LIN {X 0.032,Y -167.550,Z 313.355,A 0.000,B 0.000,C 90.000,E1 243.896} C_DIS
LIN {X 0.046,Y -166.172,Z 313.345,A 0.000,B 0.000,C 90.000,E1 242.153} C_DIS
LIN {X 0.036,Y -162.944,Z 313.326,A 0.000,B 0.000,C 90.000,E1 238.663} C_DIS
LIN {X 0.014,Y -161.614,Z 313.316,A 0.000,B 0.000,C 90.000,E1 236.914} C_DIS
LIN {X -0.011,Y -159.142,Z 313.302,A 0.000,B 0.000,C 90.000,E1 234.276} C_DIS
LIN {X -0.001,Y -155.664,Z 313.277,A 0.000,B 0.000,C 90.000,E1 229.828} C_DIS
LIN {X 0.052,Y -151.932,Z 313.252,A 0.000,B 0.000,C 90.000,E1 225.324} C_DIS
LIN {X 0.066,Y -150.169,Z 313.237,A 0.000,B 0.000,C 90.000,E1 222.609} C_DIS
LIN {X -0.014,Y -146.946,Z 313.212,A 0.000,B 0.000,C 90.000,E1 218.096} C_DIS
LIN {X -0.026,Y -145.534,Z 313.196,A 0.000,B 0.000,C 90.000,E1 215.358} C_DIS
LIN {X 0.014,Y -142.931,Z 313.171,A 0.000,B 0.000,C 90.000,E1 210.747} C_DIS
LIN {X 0.013,Y -141.555,Z 313.150,A 0.000,B 0.000,C 90.000,E1 207.052} C_DIS
LIN {X 0.001,Y -139.407,Z 313.114,A 0.000,B 0.000,C 90.000,E1 200.556} C_DIS
LIN {X -0.077,Y -139.126,Z 313.104,A 0.000,B 0.000,C 90.000,E1 198.725} C_DIS
LIN {X -0.050,Y -138.351,Z 313.057,A 0.000,B 0.000,C 90.000,E1 190.310} C_DIS
LIN {X -0.062,Y -139.500,Z 313.005,A 0.000,B 0.000,C 90.000,E1 180.974} C_DIS
LIN {X 0.018,Y -141.125,Z 312.974,A 0.000,B 0.000,C 90.000,E1 175.355} C_DIS
LIN {X -0.029,Y -142.505,Z 312.959,A 0.000,B 0.000,C 90.000,E1 172.591} C_DIS
LIN {X 0.059,Y -144.762,Z 312.933,A 0.000,B 0.000,C 90.000,E1 167.937} C_DIS
LIN {X 0.008,Y -147.373,Z 312.913,A 0.000,B 0.000,C 90.000,E1 164.283} C_DIS
LIN {X 0.071,Y -150.702,Z 312.887,A 0.000,B 0.000,C 90.000,E1 159.699} C_DIS
LIN {X 0.013,Y -154.182,Z 312.867,A 0.000,B 0.000,C 90.000,E1 156.102} C_DIS
LIN {X -0.058,Y -157.618,Z 312.847,A 0.000,B 0.000,C 90.000,E1 152.538} C_DIS
LIN {X 0.030,Y -161.873,Z 312.828,A 0.000,B 0.000,C 90.000,E1 148.948} C_DIS
LIN {X 0.003,Y -166.064,Z 312.808,A 0.000,B 0.000,C 90.000,E1 145.435} C_DIS
LIN {X 0.004,Y -171.069,Z 312.789,A 0.000,B 0.000,C 90.000,E1 141.949} C_DIS
LIN {X 0.060,Y -175.942,Z 312.769,A 0.000,B 0.000,C 90.000,E1 138.485} C_DIS
LIN {X -0.080,Y -180.183,Z 312.755,A 0.000,B 0.000,C 90.000,E1 135.972} C_DIS
LIN {X -0.112,Y -185.599,Z 312.737,A 0.000,B 0.000,C 90.000,E1 132.609} C_DIS
LIN {X -0.062,Y -190.191,Z 312.723,A 0.000,B 0.000,C 90.000,E1 130.092} C_DIS
LIN {X -0.018,Y -197.520,Z 312.700,A 0.000,B 0.000,C 90.000,E1 125.964} C_DIS
LIN {X -0.040,Y -201.256,Z 312.689,A 0.000,B 0.000,C 90.000,E1 124.072} C_DIS
LIN {X 0.037,Y -201.982,Z 312.687,A 0.000,B 0.000,C 90.000,E1 123.627} C_DIS
LIN {X 0.021,Y -303.002,Z 312.687,A 0.000,B 0.000,C 90.000,E1 123.627} C_DIS
LIN {X 0.128,Y -307.334,Z 312.686,A 0.000,B 0.000,C 90.000,E1 123.499} C_DIS
LIN {X 0.193,Y -310.491,Z 312.685,A 0.000,B 0.000,C 90.000,E1 123.293} C_DIS
LIN {X -0.027,Y -314.159,Z 312.683,A 0.000,B 0.000,C 90.000,E1 122.959} C_DIS
LIN {X -0.196,Y -317.653,Z 312.680,A 0.000,B 0.000,C 90.000,E1 122.418} C_DIS
LIN {X -0.068,Y -320.195,Z 312.676,A 0.000,B 0.000,C 90.000,E1 121.750} C_DIS
LIN {X 0.051,Y -331.214,Z 312.660,A 0.000,B 0.000,C 90.000,E1 118.871} C_DIS
LIN {X -0.163,Y -343.646,Z 312.645,A 0.000,B 0.000,C 90.000,E1 116.104} C_DIS
LIN {X -0.044,Y -355.971,Z 312.631,A 0.000,B 0.000,C 90.000,E1 113.643} C_DIS
LIN {X 0.113,Y -369.589,Z 312.618,A 0.000,B 0.000,C 90.000,E1 111.227} C_DIS
LIN {X 0.003,Y -384.601,Z 312.605,A 0.000,B 0.000,C 90.000,E1 108.906} C_DIS
LIN {X 0.015,Y -401.116,Z 312.592,A 0.000,B 0.000,C 90.000,E1 106.622} C_DIS
LIN {X -0.074,Y -419.259,Z 312.580,A 0.000,B 0.000,C 90.000,E1 104.411} C_DIS
LIN {X 0.118,Y -438.973,Z 312.568,A 0.000,B 0.000,C 90.000,E1 102.243} C_DIS
LIN {X -0.205,Y -459.388,Z 312.557,A 0.000,B 0.000,C 90.000,E1 100.310} C_DIS
LIN {X -0.132,Y -482.952,Z 312.546,A 0.000,B 0.000,C 90.000,E1 98.276} C_DIS
LIN {X -0.206,Y -496.291,Z 312.540,A 0.000,B 0.000,C 90.000,E1 97.239} C_DIS
LIN {X 0.248,Y -500.118,Z 312.538,A 0.000,B 0.000,C 90.000,E1 96.777} C_DIS
LIN {X 0.104,Y -501.638,Z 312.536,A 0.000,B 0.000,C 90.000,E1 96.549} C_DIS
LIN {X 0.015,Y -502.770,Z 312.535,A 0.000,B 0.000,C 90.000,E1 96.315} C_DIS
LIN {X -0.190,Y -504.107,Z 312.532,A 0.000,B 0.000,C 90.000,E1 95.853} C_DIS
LIN {X 0.111,Y -504.399,Z 312.530,A 0.000,B 0.000,C 90.000,E1 95.334} C_DIS
LIN {X -0.127,Y -503.685,Z 312.527,A 0.000,B 0.000,C 90.000,E1 94.878} C_DIS
LIN {X 0.184,Y -501.840,Z 312.524,A 0.000,B 0.000,C 90.000,E1 94.359} C_DIS
LIN {X 0.067,Y -500.376,Z 312.523,A 0.000,B 0.000,C 90.000,E1 94.131} C_DIS
LIN {X 0.233,Y -494.896,Z 312.519,A 0.000,B 0.000,C 90.000,E1 93.383} C_DIS
LIN {X 0.203,Y -486.911,Z 312.514,A 0.000,B 0.000,C 90.000,E1 92.407} C_DIS
LIN {X -0.144,Y -470.368,Z 312.502,A 0.000,B 0.000,C 90.000,E1 90.458} C_DIS
LIN {X -0.142,Y -452.916,Z 312.490,A 0.000,B 0.000,C 90.000,E1 88.165} C_DIS
LIN {X -0.215,Y -433.634,Z 312.474,A 0.000,B 0.000,C 90.000,E1 85.298} C_DIS
LIN {X -0.040,Y -417.883,Z 312.459,A 0.000,B 0.000,C 90.000,E1 82.591} C_DIS
LIN {X -0.043,Y -401.966,Z 312.442,A 0.000,B 0.000,C 90.000,E1 79.567} C_DIS
LIN {X -0.004,Y -393.299,Z 312.433,A 0.000,B 0.000,C 90.000,E1 77.881} C_DIS
LIN {X 0.077,Y -383.145,Z 312.422,A 0.000,B 0.000,C 90.000,E1 75.880} C_DIS
LIN {X 0.033,Y -373.060,Z 312.410,A 0.000,B 0.000,C 90.000,E1 73.866} C_DIS
LIN {X -0.005,Y -362.935,Z 312.399,A 0.000,B 0.000,C 90.000,E1 71.819} C_DIS
LIN {X -0.135,Y -352.792,Z 312.387,A 0.000,B 0.000,C 90.000,E1 69.752} C_DIS
LIN {X 0.130,Y -338.681,Z 312.370,A 0.000,B 0.000,C 90.000,E1 66.666} C_DIS
LIN {X -0.005,Y -328.630,Z 312.357,A 0.000,B 0.000,C 90.000,E1 64.204} C_DIS
LIN {X -0.086,Y -319.293,Z 312.343,A 0.000,B 0.000,C 90.000,E1 61.691} C_DIS
LIN {X -0.033,Y -309.202,Z 312.327,A 0.000,B 0.000,C 90.000,E1 58.791} C_DIS
LIN {X -0.003,Y -298.551,Z 312.308,A 0.000,B 0.000,C 90.000,E1 55.515} C_DIS
LIN {X 0.062,Y -290.540,Z 312.294,A 0.000,B 0.000,C 90.000,E1 52.844} C_DIS
LIN {X 0.038,Y -282.742,Z 312.279,A 0.000,B 0.000,C 90.000,E1 50.150} C_DIS
LIN {X 0.136,Y -276.853,Z 312.267,A 0.000,B 0.000,C 90.000,E1 48.081} C_DIS
LIN {X 0.082,Y -269.108,Z 312.252,A 0.000,B 0.000,C 90.000,E1 45.324} C_DIS
LIN {X 0.023,Y -261.659,Z 312.236,A 0.000,B 0.000,C 90.000,E1 42.528} C_DIS
LIN {X 0.102,Y -255.970,Z 312.224,A 0.000,B 0.000,C 90.000,E1 40.378} C_DIS
LIN {X -0.058,Y -250.303,Z 312.212,A 0.000,B 0.000,C 90.000,E1 38.257} C_DIS
LIN {X -0.119,Y -244.496,Z 312.200,A 0.000,B 0.000,C 90.000,E1 36.091} C_DIS
LIN {X -0.035,Y -238.536,Z 312.188,A 0.000,B 0.000,C 90.000,E1 33.865} C_DIS
LIN {X -0.008,Y -230.819,Z 312.172,A 0.000,B 0.000,C 90.000,E1 30.875} C_DIS
LIN {X -0.016,Y -223.411,Z 312.155,A 0.000,B 0.000,C 90.000,E1 27.847} C_DIS
LIN {X -0.021,Y -216.773,Z 312.138,A 0.000,B 0.000,C 90.000,E1 24.771} C_DIS
LIN {X -0.064,Y -210.982,Z 312.120,A 0.000,B 0.000,C 90.000,E1 21.663} C_DIS
LIN {X -0.005,Y -205.942,Z 312.103,A 0.000,B 0.000,C 90.000,E1 18.489} C_DIS
LIN {X -0.016,Y -201.693,Z 312.085,A 0.000,B 0.000,C 90.000,E1 15.300} C_DIS
LIN {X 0.077,Y -197.331,Z 312.063,A 0.000,B 0.000,C 90.000,E1 11.243} C_DIS
LIN {X 0.052,Y -193.957,Z 312.040,A 0.000,B 0.000,C 90.000,E1 7.182} C_DIS
LIN {X 0.080,Y -190.978,Z 312.008,A 0.000,B 0.000,C 90.000,E1 1.432} C_DIS
LIN {X -0.060,Y -192.059,Z 311.929,A 0.000,B 0.000,C 90.000,E1 347.173} C_DIS
LIN {X -0.012,Y -195.378,Z 311.901,A 0.000,B 0.000,C 90.000,E1 342.236} C_DIS
LIN {X 0.012,Y -199.257,Z 311.879,A 0.000,B 0.000,C 90.000,E1 338.156} C_DIS
LIN {X -0.101,Y -204.157,Z 311.856,A 0.000,B 0.000,C 90.000,E1 334.152} C_DIS
LIN {X 0.022,Y -210.144,Z 311.834,A 0.000,B 0.000,C 90.000,E1 330.127} C_DIS
LIN {X -0.075,Y -216.868,Z 311.812,A 0.000,B 0.000,C 90.000,E1 326.215} C_DIS
LIN {X 0.004,Y -222.927,Z 311.795,A 0.000,B 0.000,C 90.000,E1 323.084} C_DIS
LIN {X 0.108,Y -229.781,Z 311.778,A 0.000,B 0.000,C 90.000,E1 319.989} C_DIS
LIN {X 0.027,Y -237.717,Z 311.761,A 0.000,B 0.000,C 90.000,E1 316.986} C_DIS
LIN {X -0.018,Y -246.728,Z 311.745,A 0.000,B 0.000,C 90.000,E1 314.028} C_DIS
LIN {X 0.023,Y -257.971,Z 311.726,A 0.000,B 0.000,C 90.000,E1 310.744} C_DIS
LIN {X 0.113,Y -270.170,Z 311.709,A 0.000,B 0.000,C 90.000,E1 307.523} C_DIS
LIN {X 0.083,Y -283.606,Z 311.691,A 0.000,B 0.000,C 90.000,E1 304.405} C_DIS
LIN {X -0.043,Y -295.197,Z 311.678,A 0.000,B 0.000,C 90.000,E1 302.054} C_DIS
LIN {X -0.057,Y -311.692,Z 311.661,A 0.000,B 0.000,C 90.000,E1 299.077} C_DIS
LIN {X 0.023,Y -327.977,Z 311.647,A 0.000,B 0.000,C 90.000,E1 296.488} C_DIS
LIN {X 0.098,Y -343.187,Z 311.635,A 0.000,B 0.000,C 90.000,E1 294.283} C_DIS
LIN {X 0.064,Y -358.770,Z 311.623,A 0.000,B 0.000,C 90.000,E1 292.153} C_DIS
LIN {X 0.087,Y -374.576,Z 311.612,A 0.000,B 0.000,C 90.000,E1 290.066} C_DIS
LIN {X 0.158,Y -395.796,Z 311.597,A 0.000,B 0.000,C 90.000,E1 287.457} C_DIS
LIN {X 0.037,Y -410.146,Z 311.588,A 0.000,B 0.000,C 90.000,E1 285.788} C_DIS
LIN {X 0.028,Y -422.019,Z 311.580,A 0.000,B 0.000,C 90.000,E1 284.411} C_DIS
LIN {X -0.188,Y -431.113,Z 311.574,A 0.000,B 0.000,C 90.000,E1 283.355} C_DIS
LIN {X -0.061,Y -437.406,Z 311.570,A 0.000,B 0.000,C 90.000,E1 282.535} C_DIS
LIN {X -0.094,Y -445.195,Z 311.564,A 0.000,B 0.000,C 90.000,E1 281.478} C_DIS
LIN {X -0.039,Y -452.384,Z 311.558,A 0.000,B 0.000,C 90.000,E1 280.423} C_DIS
LIN {X -0.241,Y -460.518,Z 311.551,A 0.000,B 0.000,C 90.000,E1 279.151} C_DIS
LIN {X 0.214,Y -467.942,Z 311.544,A 0.000,B 0.000,C 90.000,E1 277.814} C_DIS
LIN {X 0.189,Y -474.932,Z 311.536,A 0.000,B 0.000,C 90.000,E1 276.549} C_DIS
LIN {X -0.016,Y -479.846,Z 311.531,A 0.000,B 0.000,C 90.000,E1 275.568} C_DIS
LIN {X 0.139,Y -481.878,Z 311.528,A 0.000,B 0.000,C 90.000,E1 275.049} C_DIS
LIN {X -0.181,Y -483.529,Z 311.525,A 0.000,B 0.000,C 90.000,E1 274.588} C_DIS
LIN {X -0.046,Y -484.766,Z 311.523,A 0.000,B 0.000,C 90.000,E1 274.073} C_DIS
LIN {X 0.136,Y -485.673,Z 311.520,A 0.000,B 0.000,C 90.000,E1 273.555} C_DIS
LIN {X -0.165,Y -486.197,Z 311.517,A 0.000,B 0.000,C 90.000,E1 273.094} C_DIS
LIN {X -0.001,Y -486.339,Z 311.514,A 0.000,B 0.000,C 90.000,E1 272.579} C_DIS
LIN {X 0.169,Y -486.185,Z 311.512,A 0.000,B 0.000,C 90.000,E1 272.064} C_DIS
LIN {X -0.129,Y -485.840,Z 311.509,A 0.000,B 0.000,C 90.000,E1 271.604} C_DIS
LIN {X 0.211,Y -484.662,Z 311.503,A 0.000,B 0.000,C 90.000,E1 270.573} C_DIS
LIN {X -0.107,Y -483.765,Z 311.501,A 0.000,B 0.000,C 90.000,E1 270.115} C_DIS
LIN {X 0.056,Y -482.489,Z 311.498,A 0.000,B 0.000,C 90.000,E1 269.599} C_DIS
LIN {X 0.213,Y -480.691,Z 311.495,A 0.000,B 0.000,C 90.000,E1 269.083} C_DIS
LIN {X -0.118,Y -478.303,Z 311.492,A 0.000,B 0.000,C 90.000,E1 268.625} C_DIS
LIN {X 0.027,Y -475.065,Z 311.490,A 0.000,B 0.000,C 90.000,E1 268.108} C_DIS
LIN {X -0.152,Y -473.122,Z 311.488,A 0.000,B 0.000,C 90.000,E1 267.879} C_DIS
LIN {X -0.049,Y -468.280,Z 311.485,A 0.000,B 0.000,C 90.000,E1 267.364} C_DIS
LIN {X -0.238,Y -465.410,Z 311.484,A 0.000,B 0.000,C 90.000,E1 267.135} C_DIS
LIN {X -0.234,Y -462.356,Z 311.483,A 0.000,B 0.000,C 90.000,E1 266.906} C_DIS
LIN {X -0.205,Y -458.818,Z 311.481,A 0.000,B 0.000,C 90.000,E1 266.674} C_DIS
LIN {X 0.159,Y -455.570,Z 311.480,A 0.000,B 0.000,C 90.000,E1 266.445} C_DIS
LIN {X -0.165,Y -448.436,Z 311.479,A 0.000,B 0.000,C 90.000,E1 266.159} C_DIS
LIN {X 0.055,Y -444.407,Z 311.478,A 0.000,B 0.000,C 90.000,E1 265.988} C_DIS
LIN {X 0.153,Y -436.095,Z 311.477,A 0.000,B 0.000,C 90.000,E1 265.755} C_DIS
LIN {X 0.129,Y -428.549,Z 311.476,A 0.000,B 0.000,C 90.000,E1 265.641} C_DIS
LIN {X -0.013,Y -417.647,Z 311.475,A 0.000,B 0.000,C 90.000,E1 265.584} C_DIS
LIN {X -0.035,Y -180.908,Z 311.475,A 0.000,B 0.000,C 90.000,E1 265.584} C_DIS
LIN {X -0.045,Y -180.691,Z 311.470,A 0.000,B 0.000,C 90.000,E1 264.546} C_DIS
LIN {X -0.037,Y -179.027,Z 311.445,A 0.000,B 0.000,C 90.000,E1 260.151} C_DIS
LIN {X 0.026,Y -178.671,Z 311.441,A 0.000,B 0.000,C 90.000,E1 259.285} C_DIS
LIN {X -0.039,Y -175.721,Z 311.412,A 0.000,B 0.000,C 90.000,E1 254.212} C_DIS
LIN {X -0.022,Y -172.437,Z 311.388,A 0.000,B 0.000,C 90.000,E1 249.934} C_DIS
LIN {X -0.067,Y -171.267,Z 311.379,A 0.000,B 0.000,C 90.000,E1 248.230} C_DIS
LIN {X -0.021,Y -167.537,Z 311.355,A 0.000,B 0.000,C 90.000,E1 243.896} C_DIS
LIN {X -0.007,Y -166.152,Z 311.345,A 0.000,B 0.000,C 90.000,E1 242.153} C_DIS
LIN {X -0.016,Y -162.929,Z 311.326,A 0.000,B 0.000,C 90.000,E1 238.663} C_DIS
LIN {X -0.038,Y -161.601,Z 311.316,A 0.000,B 0.000,C 90.000,E1 236.914} C_DIS
LIN {X 0.087,Y -158.345,Z 311.296,A 0.000,B 0.000,C 90.000,E1 233.336} C_DIS
LIN {X -0.052,Y -155.647,Z 311.277,A 0.000,B 0.000,C 90.000,E1 229.828} C_DIS
LIN {X 0.001,Y -151.919,Z 311.252,A 0.000,B 0.000,C 90.000,E1 225.324} C_DIS
LIN {X 0.017,Y -150.153,Z 311.237,A 0.000,B 0.000,C 90.000,E1 222.609} C_DIS
LIN {X -0.063,Y -146.935,Z 311.212,A 0.000,B 0.000,C 90.000,E1 218.096} C_DIS
LIN {X 0.044,Y -145.523,Z 311.196,A 0.000,B 0.000,C 90.000,E1 215.311} C_DIS
LIN {X 0.039,Y -142.922,Z 311.171,A 0.000,B 0.000,C 90.000,E1 210.718} C_DIS
LIN {X -0.035,Y -141.546,Z 311.150,A 0.000,B 0.000,C 90.000,E1 207.052} C_DIS
LIN {X -0.046,Y -139.404,Z 311.114,A 0.000,B 0.000,C 90.000,E1 200.556} C_DIS
LIN {X 0.008,Y -139.121,Z 311.104,A 0.000,B 0.000,C 90.000,E1 198.671} C_DIS
LIN {X 0.039,Y -138.352,Z 311.057,A 0.000,B 0.000,C 90.000,E1 190.254} C_DIS
LIN {X 0.029,Y -139.502,Z 311.005,A 0.000,B 0.000,C 90.000,E1 180.917} C_DIS
LIN {X -0.030,Y -141.133,Z 310.974,A 0.000,B 0.000,C 90.000,E1 175.355} C_DIS
LIN {X -0.077,Y -142.514,Z 310.959,A 0.000,B 0.000,C 90.000,E1 172.591} C_DIS
LIN {X 0.010,Y -144.774,Z 310.933,A 0.000,B 0.000,C 90.000,E1 167.937} C_DIS
LIN {X -0.041,Y -147.388,Z 310.913,A 0.000,B 0.000,C 90.000,E1 164.283} C_DIS
LIN {X 0.022,Y -150.718,Z 310.887,A 0.000,B 0.000,C 90.000,E1 159.699} C_DIS
LIN {X -0.038,Y -154.199,Z 310.867,A 0.000,B 0.000,C 90.000,E1 156.102} C_DIS
LIN {X 0.030,Y -157.638,Z 310.847,A 0.000,B 0.000,C 90.000,E1 152.487} C_DIS
LIN {X -0.022,Y -161.896,Z 310.827,A 0.000,B 0.000,C 90.000,E1 148.948} C_DIS
LIN {X 0.087,Y -166.087,Z 310.808,A 0.000,B 0.000,C 90.000,E1 145.388} C_DIS
LIN {X 0.085,Y -171.094,Z 310.789,A 0.000,B 0.000,C 90.000,E1 141.904} C_DIS
LIN {X 0.006,Y -175.969,Z 310.769,A 0.000,B 0.000,C 90.000,E1 138.485} C_DIS
LIN {X 0.120,Y -180.214,Z 310.755,A 0.000,B 0.000,C 90.000,E1 135.891} C_DIS
LIN {X 0.095,Y -185.629,Z 310.736,A 0.000,B 0.000,C 90.000,E1 132.528} C_DIS
LIN {X -0.119,Y -190.225,Z 310.723,A 0.000,B 0.000,C 90.000,E1 130.092} C_DIS
LIN {X 0.039,Y -197.554,Z 310.700,A 0.000,B 0.000,C 90.000,E1 125.931} C_DIS
LIN {X 0.012,Y -201.285,Z 310.689,A 0.000,B 0.000,C 90.000,E1 124.040} C_DIS
LIN {X 0.072,Y -202.049,Z 310.687,A 0.000,B 0.000,C 90.000,E1 123.579} C_DIS
LIN {X 0.073,Y -303.497,Z 310.687,A 0.000,B 0.000,C 90.000,E1 123.579} C_DIS
LIN {X -0.033,Y -304.873,Z 310.687,A 0.000,B 0.000,C 90.000,E1 123.579} C_DIS
LIN {X 0.038,Y -307.008,Z 310.686,A 0.000,B 0.000,C 90.000,E1 123.499} C_DIS
LIN {X 0.095,Y -310.374,Z 310.685,A 0.000,B 0.000,C 90.000,E1 123.293} C_DIS
LIN {X -0.025,Y -313.978,Z 310.683,A 0.000,B 0.000,C 90.000,E1 122.959} C_DIS
LIN {X -0.112,Y -317.508,Z 310.680,A 0.000,B 0.000,C 90.000,E1 122.418} C_DIS
LIN {X -0.048,Y -318.945,Z 310.678,A 0.000,B 0.000,C 90.000,E1 122.084} C_DIS
LIN {X 0.136,Y -331.133,Z 310.661,A 0.000,B 0.000,C 90.000,E1 118.871} C_DIS
LIN {X -0.077,Y -343.556,Z 310.645,A 0.000,B 0.000,C 90.000,E1 116.104} C_DIS
LIN {X 0.041,Y -355.873,Z 310.631,A 0.000,B 0.000,C 90.000,E1 113.643} C_DIS
LIN {X -0.145,Y -369.484,Z 310.618,A 0.000,B 0.000,C 90.000,E1 111.280} C_DIS
LIN {X 0.089,Y -384.487,Z 310.605,A 0.000,B 0.000,C 90.000,E1 108.906} C_DIS
LIN {X 0.103,Y -400.993,Z 310.592,A 0.000,B 0.000,C 90.000,E1 106.622} C_DIS
LIN {X 0.015,Y -419.126,Z 310.580,A 0.000,B 0.000,C 90.000,E1 104.411} C_DIS
LIN {X -0.224,Y -438.833,Z 310.568,A 0.000,B 0.000,C 90.000,E1 102.299} C_DIS
LIN {X -0.123,Y -459.245,Z 310.557,A 0.000,B 0.000,C 90.000,E1 100.310} C_DIS
LIN {X -0.055,Y -482.807,Z 310.546,A 0.000,B 0.000,C 90.000,E1 98.276} C_DIS
LIN {X -0.131,Y -496.163,Z 310.540,A 0.000,B 0.000,C 90.000,E1 97.239} C_DIS
LIN {X -0.157,Y -500.131,Z 310.538,A 0.000,B 0.000,C 90.000,E1 96.834} C_DIS
LIN {X 0.195,Y -501.711,Z 310.536,A 0.000,B 0.000,C 90.000,E1 96.549} C_DIS
LIN {X 0.106,Y -502.893,Z 310.535,A 0.000,B 0.000,C 90.000,E1 96.315} C_DIS
LIN {X -0.099,Y -504.306,Z 310.532,A 0.000,B 0.000,C 90.000,E1 95.853} C_DIS
LIN {X 0.203,Y -504.662,Z 310.530,A 0.000,B 0.000,C 90.000,E1 95.334} C_DIS
LIN {X -0.034,Y -504.015,Z 310.527,A 0.000,B 0.000,C 90.000,E1 94.878} C_DIS
LIN {X -0.223,Y -502.249,Z 310.524,A 0.000,B 0.000,C 90.000,E1 94.416} C_DIS
LIN {X 0.161,Y -500.840,Z 310.523,A 0.000,B 0.000,C 90.000,E1 94.131} C_DIS
LIN {X -0.164,Y -495.358,Z 310.519,A 0.000,B 0.000,C 90.000,E1 93.440} C_DIS
LIN {X -0.183,Y -487.383,Z 310.514,A 0.000,B 0.000,C 90.000,E1 92.465} C_DIS
LIN {X -0.035,Y -470.808,Z 310.503,A 0.000,B 0.000,C 90.000,E1 90.458} C_DIS
LIN {X -0.027,Y -453.301,Z 310.490,A 0.000,B 0.000,C 90.000,E1 88.165} C_DIS
LIN {X 0.181,Y -435.674,Z 310.475,A 0.000,B 0.000,C 90.000,E1 85.527} C_DIS
LIN {X -0.162,Y -421.238,Z 310.462,A 0.000,B 0.000,C 90.000,E1 83.166} C_DIS
LIN {X -0.010,Y -403.704,Z 310.444,A 0.000,B 0.000,C 90.000,E1 79.859} C_DIS
LIN {X -0.020,Y -396.561,Z 310.436,A 0.000,B 0.000,C 90.000,E1 78.465} C_DIS
LIN {X 0.175,Y -384.928,Z 310.423,A 0.000,B 0.000,C 90.000,E1 76.172} C_DIS
LIN {X -0.183,Y -373.391,Z 310.411,A 0.000,B 0.000,C 90.000,E1 73.921} C_DIS
LIN {X 0.140,Y -363.278,Z 310.399,A 0.000,B 0.000,C 90.000,E1 71.819} C_DIS
LIN {X 0.061,Y -351.733,Z 310.386,A 0.000,B 0.000,C 90.000,E1 69.444} C_DIS
LIN {X -0.022,Y -337.752,Z 310.369,A 0.000,B 0.000,C 90.000,E1 66.410} C_DIS
LIN {X -0.149,Y -324.302,Z 310.350,A 0.000,B 0.000,C 90.000,E1 62.999} C_DIS
LIN {X -0.115,Y -313.999,Z 310.334,A 0.000,B 0.000,C 90.000,E1 60.127} C_DIS
LIN {X -0.186,Y -307.371,Z 310.323,A 0.000,B 0.000,C 90.000,E1 58.201} C_DIS
LIN {X -0.041,Y -296.873,Z 310.305,A 0.000,B 0.000,C 90.000,E1 54.895} C_DIS
LIN {X 0.153,Y -288.917,Z 310.290,A 0.000,B 0.000,C 90.000,E1 52.190} C_DIS
LIN {X 0.003,Y -283.059,Z 310.279,A 0.000,B 0.000,C 90.000,E1 50.194} C_DIS
LIN {X -0.071,Y -277.165,Z 310.267,A 0.000,B 0.000,C 90.000,E1 48.162} C_DIS
LIN {X -0.113,Y -269.385,Z 310.252,A 0.000,B 0.000,C 90.000,E1 45.405} C_DIS
LIN {X -0.159,Y -261.943,Z 310.237,A 0.000,B 0.000,C 90.000,E1 42.609} C_DIS
LIN {X -0.071,Y -256.269,Z 310.225,A 0.000,B 0.000,C 90.000,E1 40.458} C_DIS
LIN {X -0.023,Y -248.705,Z 310.209,A 0.000,B 0.000,C 90.000,E1 37.569} C_DIS
LIN {X -0.066,Y -242.824,Z 310.197,A 0.000,B 0.000,C 90.000,E1 35.391} C_DIS
LIN {X -0.001,Y -234.927,Z 310.180,A 0.000,B 0.000,C 90.000,E1 32.418} C_DIS
LIN {X 0.008,Y -227.302,Z 310.163,A 0.000,B 0.000,C 90.000,E1 29.411} C_DIS
LIN {X 0.002,Y -220.309,Z 310.146,A 0.000,B 0.000,C 90.000,E1 26.360} C_DIS
LIN {X 0.018,Y -214.034,Z 310.129,A 0.000,B 0.000,C 90.000,E1 23.259} C_DIS
LIN {X 0.020,Y -208.675,Z 310.112,A 0.000,B 0.000,C 90.000,E1 20.120} C_DIS
LIN {X -0.057,Y -204.012,Z 310.094,A 0.000,B 0.000,C 90.000,E1 16.968} C_DIS
LIN {X 0.008,Y -199.226,Z 310.072,A 0.000,B 0.000,C 90.000,E1 12.939} C_DIS
LIN {X -0.090,Y -195.395,Z 310.049,A 0.000,B 0.000,C 90.000,E1 8.916} C_DIS
LIN {X 0.036,Y -191.837,Z 310.018,A 0.000,B 0.000,C 90.000,E1 3.154} C_DIS
LIN {X -0.052,Y -192.644,Z 309.924,A 0.000,B 0.000,C 90.000,E1 346.353} C_DIS
LIN {X 0.066,Y -196.203,Z 309.897,A 0.000,B 0.000,C 90.000,E1 341.402} C_DIS
LIN {X -0.005,Y -200.258,Z 309.874,A 0.000,B 0.000,C 90.000,E1 337.358} C_DIS
LIN {X -0.008,Y -205.355,Z 309.852,A 0.000,B 0.000,C 90.000,E1 333.332} C_DIS
LIN {X 0.070,Y -211.486,Z 309.830,A 0.000,B 0.000,C 90.000,E1 329.331} C_DIS
LIN {X 0.135,Y -218.377,Z 309.808,A 0.000,B 0.000,C 90.000,E1 325.388} C_DIS
LIN {X 0.032,Y -224.624,Z 309.791,A 0.000,B 0.000,C 90.000,E1 322.316} C_DIS
LIN {X 0.041,Y -231.765,Z 309.774,A 0.000,B 0.000,C 90.000,E1 319.256} C_DIS
LIN {X -0.029,Y -241.098,Z 309.755,A 0.000,B 0.000,C 90.000,E1 315.891} C_DIS
LIN {X -0.164,Y -251.768,Z 309.737,A 0.000,B 0.000,C 90.000,E1 312.609} C_DIS
LIN {X 0.041,Y -263.397,Z 309.719,A 0.000,B 0.000,C 90.000,E1 309.322} C_DIS
LIN {X -0.038,Y -276.135,Z 309.701,A 0.000,B 0.000,C 90.000,E1 306.171} C_DIS
LIN {X -0.038,Y -288.608,Z 309.686,A 0.000,B 0.000,C 90.000,E1 303.420} C_DIS
LIN {X 0.037,Y -300.736,Z 309.673,A 0.000,B 0.000,C 90.000,E1 301.052} C_DIS
LIN {X 0.037,Y -317.853,Z 309.656,A 0.000,B 0.000,C 90.000,E1 298.103} C_DIS
LIN {X -0.191,Y -336.869,Z 309.640,A 0.000,B 0.000,C 90.000,E1 295.283} C_DIS
LIN {X 0.078,Y -352.288,Z 309.628,A 0.000,B 0.000,C 90.000,E1 293.078} C_DIS
LIN {X 0.021,Y -365.734,Z 309.618,A 0.000,B 0.000,C 90.000,E1 291.280} C_DIS
LIN {X -0.043,Y -386.328,Z 309.604,A 0.000,B 0.000,C 90.000,E1 288.652} C_DIS
LIN {X 0.150,Y -400.658,Z 309.594,A 0.000,B 0.000,C 90.000,E1 286.913} C_DIS
LIN {X 0.114,Y -414.908,Z 309.585,A 0.000,B 0.000,C 90.000,E1 285.245} C_DIS
LIN {X 0.068,Y -426.606,Z 309.577,A 0.000,B 0.000,C 90.000,E1 283.883} C_DIS
LIN {X 0.154,Y -433.207,Z 309.573,A 0.000,B 0.000,C 90.000,E1 283.063} C_DIS
LIN {X 0.077,Y -441.243,Z 309.567,A 0.000,B 0.000,C 90.000,E1 282.007} C_DIS
LIN {X 0.090,Y -448.733,Z 309.561,A 0.000,B 0.000,C 90.000,E1 280.950} C_DIS
LIN {X 0.108,Y -455.550,Z 309.555,A 0.000,B 0.000,C 90.000,E1 279.905} C_DIS
LIN {X 0.207,Y -461.857,Z 309.549,A 0.000,B 0.000,C 90.000,E1 278.859} C_DIS
LIN {X 0.155,Y -469.202,Z 309.542,A 0.000,B 0.000,C 90.000,E1 277.587} C_DIS
LIN {X -0.116,Y -474.739,Z 309.537,A 0.000,B 0.000,C 90.000,E1 276.606} C_DIS
LIN {X -0.134,Y -478.477,Z 309.532,A 0.000,B 0.000,C 90.000,E1 275.853} C_DIS
LIN {X -0.174,Y -481.677,Z 309.528,A 0.000,B 0.000,C 90.000,E1 275.106} C_DIS
LIN {X -0.015,Y -483.377,Z 309.525,A 0.000,B 0.000,C 90.000,E1 274.588} C_DIS
LIN {X 0.119,Y -484.669,Z 309.523,A 0.000,B 0.000,C 90.000,E1 274.073} C_DIS
LIN {X -0.184,Y -485.581,Z 309.520,A 0.000,B 0.000,C 90.000,E1 273.612} C_DIS
LIN {X 0.000,Y -486.111,Z 309.517,A 0.000,B 0.000,C 90.000,E1 273.094} C_DIS
LIN {X 0.163,Y -486.287,Z 309.514,A 0.000,B 0.000,C 90.000,E1 272.579} C_DIS
LIN {X 0.033,Y -485.797,Z 309.509,A 0.000,B 0.000,C 90.000,E1 271.604} C_DIS
LIN {X -0.113,Y -484.633,Z 309.503,A 0.000,B 0.000,C 90.000,E1 270.630} C_DIS
LIN {X 0.054,Y -483.779,Z 309.501,A 0.000,B 0.000,C 90.000,E1 270.115} C_DIS
LIN {X 0.218,Y -482.554,Z 309.498,A 0.000,B 0.000,C 90.000,E1 269.599} C_DIS
LIN {X -0.108,Y -480.815,Z 309.495,A 0.000,B 0.000,C 90.000,E1 269.141} C_DIS
LIN {X 0.042,Y -478.459,Z 309.492,A 0.000,B 0.000,C 90.000,E1 268.625} C_DIS
LIN {X 0.186,Y -475.265,Z 309.490,A 0.000,B 0.000,C 90.000,E1 268.108} C_DIS
LIN {X 0.007,Y -473.353,Z 309.488,A 0.000,B 0.000,C 90.000,E1 267.879} C_DIS
LIN {X -0.171,Y -471.137,Z 309.487,A 0.000,B 0.000,C 90.000,E1 267.650} C_DIS
LIN {X -0.080,Y -465.785,Z 309.484,A 0.000,B 0.000,C 90.000,E1 267.135} C_DIS
LIN {X -0.100,Y -462.759,Z 309.483,A 0.000,B 0.000,C 90.000,E1 266.906} C_DIS
LIN {X -0.093,Y -459.276,Z 309.481,A 0.000,B 0.000,C 90.000,E1 266.674} C_DIS
LIN {X -0.217,Y -456.010,Z 309.480,A 0.000,B 0.000,C 90.000,E1 266.502} C_DIS
LIN {X -0.138,Y -448.835,Z 309.479,A 0.000,B 0.000,C 90.000,E1 266.159} C_DIS
LIN {X 0.061,Y -444.893,Z 309.478,A 0.000,B 0.000,C 90.000,E1 265.988} C_DIS
LIN {X 0.099,Y -436.344,Z 309.477,A 0.000,B 0.000,C 90.000,E1 265.755} C_DIS
LIN {X -0.048,Y -432.168,Z 309.476,A 0.000,B 0.000,C 90.000,E1 265.698} C_DIS
LIN {X -0.191,Y -425.842,Z 309.476,A 0.000,B 0.000,C 90.000,E1 265.641} C_DIS
LIN {X -0.162,Y -415.665,Z 309.475,A 0.000,B 0.000,C 90.000,E1 265.584} C_DIS
LIN {X 0.075,Y -180.907,Z 309.475,A 0.000,B 0.000,C 90.000,E1 265.527} C_DIS
LIN {X 0.065,Y -180.762,Z 309.470,A 0.000,B 0.000,C 90.000,E1 264.666} C_DIS
LIN {X -0.043,Y -178.855,Z 309.442,A 0.000,B 0.000,C 90.000,E1 259.634} C_DIS
LIN {X 0.027,Y -175.899,Z 309.414,A 0.000,B 0.000,C 90.000,E1 254.519} C_DIS
LIN {X -0.034,Y -174.577,Z 309.405,A 0.000,B 0.000,C 90.000,E1 252.834} C_DIS
LIN {X 0.003,Y -171.560,Z 309.381,A 0.000,B 0.000,C 90.000,E1 248.539} C_DIS
LIN {X 0.058,Y -167.783,Z 309.357,A 0.000,B 0.000,C 90.000,E1 244.204} C_DIS
LIN {X -0.001,Y -166.496,Z 309.347,A 0.000,B 0.000,C 90.000,E1 242.487} C_DIS
LIN {X -0.006,Y -163.207,Z 309.328,A 0.000,B 0.000,C 90.000,E1 238.997} C_DIS
LIN {X -0.040,Y -161.171,Z 309.313,A 0.000,B 0.000,C 90.000,E1 236.373} C_DIS
LIN {X 0.083,Y -157.186,Z 309.289,A 0.000,B 0.000,C 90.000,E1 231.904} C_DIS
LIN {X 0.006,Y -155.916,Z 309.279,A 0.000,B 0.000,C 90.000,E1 230.150} C_DIS
LIN {X 0.063,Y -152.166,Z 309.254,A 0.000,B 0.000,C 90.000,E1 225.648} C_DIS
LIN {X -0.028,Y -150.414,Z 309.239,A 0.000,B 0.000,C 90.000,E1 222.975} C_DIS
LIN {X 0.013,Y -147.143,Z 309.213,A 0.000,B 0.000,C 90.000,E1 218.418} C_DIS
LIN {X 0.010,Y -145.702,Z 309.198,A 0.000,B 0.000,C 90.000,E1 215.678} C_DIS
LIN {X 0.019,Y -143.085,Z 309.173,A 0.000,B 0.000,C 90.000,E1 211.082} C_DIS
LIN {X 0.023,Y -141.702,Z 309.152,A 0.000,B 0.000,C 90.000,E1 207.385} C_DIS
LIN {X -0.054,Y -139.467,Z 309.116,A 0.000,B 0.000,C 90.000,E1 200.918} C_DIS
LIN {X 0.000,Y -139.200,Z 309.106,A 0.000,B 0.000,C 90.000,E1 199.033} C_DIS
LIN {X 0.063,Y -138.328,Z 309.054,A 0.000,B 0.000,C 90.000,E1 189.670} C_DIS
LIN {X 0.068,Y -139.444,Z 309.007,A 0.000,B 0.000,C 90.000,E1 181.260} C_DIS
LIN {X 0.009,Y -140.982,Z 308.976,A 0.000,B 0.000,C 90.000,E1 175.698} C_DIS
LIN {X -0.041,Y -142.737,Z 308.956,A 0.000,B 0.000,C 90.000,E1 172.008} C_DIS
LIN {X 0.057,Y -145.128,Z 308.930,A 0.000,B 0.000,C 90.000,E1 167.353} C_DIS
LIN {X 0.051,Y -147.752,Z 308.909,A 0.000,B 0.000,C 90.000,E1 163.685} C_DIS
LIN {X -0.010,Y -150.420,Z 308.889,A 0.000,B 0.000,C 90.000,E1 160.061} C_DIS
LIN {X 0.005,Y -153.861,Z 308.869,A 0.000,B 0.000,C 90.000,E1 156.433} C_DIS
LIN {X -0.078,Y -157.272,Z 308.849,A 0.000,B 0.000,C 90.000,E1 152.871} C_DIS
LIN {X -0.001,Y -161.450,Z 308.829,A 0.000,B 0.000,C 90.000,E1 149.282} C_DIS
LIN {X 0.006,Y -165.650,Z 308.810,A 0.000,B 0.000,C 90.000,E1 145.754} C_DIS
LIN {X -0.012,Y -170.585,Z 308.790,A 0.000,B 0.000,C 90.000,E1 142.271} C_DIS
LIN {X -0.105,Y -175.463,Z 308.771,A 0.000,B 0.000,C 90.000,E1 138.852} C_DIS
LIN {X 0.011,Y -181.085,Z 308.752,A 0.000,B 0.000,C 90.000,E1 135.405} C_DIS
LIN {X 0.000,Y -186.526,Z 308.734,A 0.000,B 0.000,C 90.000,E1 132.043} C_DIS
LIN {X -0.058,Y -191.143,Z 308.720,A 0.000,B 0.000,C 90.000,E1 129.564} C_DIS
LIN {X 0.020,Y -196.944,Z 308.701,A 0.000,B 0.000,C 90.000,E1 126.251} C_DIS
LIN {X 0.056,Y -200.208,Z 308.692,A 0.000,B 0.000,C 90.000,E1 124.612} C_DIS
LIN {X -0.056,Y -202.112,Z 308.686,A 0.000,B 0.000,C 90.000,E1 123.579} C_DIS
LIN {X -0.135,Y -303.945,Z 308.686,A 0.000,B 0.000,C 90.000,E1 123.579} C_DIS
LIN {X -0.012,Y -308.244,Z 308.686,A 0.000,B 0.000,C 90.000,E1 123.420} C_DIS
LIN {X -0.058,Y -310.382,Z 308.685,A 0.000,B 0.000,C 90.000,E1 123.293} C_DIS
LIN {X 0.020,Y -313.309,Z 308.683,A 0.000,B 0.000,C 90.000,E1 123.007} C_DIS
LIN {X 0.079,Y -316.996,Z 308.680,A 0.000,B 0.000,C 90.000,E1 122.467} C_DIS
LIN {X 0.138,Y -318.567,Z 308.679,A 0.000,B 0.000,C 90.000,E1 122.133} C_DIS
LIN {X -0.191,Y -332.085,Z 308.659,A 0.000,B 0.000,C 90.000,E1 118.693} C_DIS
LIN {X 0.084,Y -344.627,Z 308.644,A 0.000,B 0.000,C 90.000,E1 115.848} C_DIS
LIN {X -0.093,Y -357.061,Z 308.630,A 0.000,B 0.000,C 90.000,E1 113.439} C_DIS
LIN {X -0.052,Y -370.796,Z 308.617,A 0.000,B 0.000,C 90.000,E1 111.046} C_DIS
LIN {X -0.137,Y -385.933,Z 308.604,A 0.000,B 0.000,C 90.000,E1 108.725} C_DIS
LIN {X -0.097,Y -402.585,Z 308.591,A 0.000,B 0.000,C 90.000,E1 106.441} C_DIS
LIN {X 0.147,Y -420.875,Z 308.579,A 0.000,B 0.000,C 90.000,E1 104.189} C_DIS
LIN {X 0.127,Y -440.673,Z 308.567,A 0.000,B 0.000,C 90.000,E1 102.063} C_DIS
LIN {X -0.167,Y -461.135,Z 308.556,A 0.000,B 0.000,C 90.000,E1 100.141} C_DIS
LIN {X 0.022,Y -484.775,Z 308.545,A 0.000,B 0.000,C 90.000,E1 98.106} C_DIS
LIN {X -0.180,Y -495.458,Z 308.540,A 0.000,B 0.000,C 90.000,E1 97.296} C_DIS
LIN {X 0.041,Y -497.914,Z 308.539,A 0.000,B 0.000,C 90.000,E1 97.068} C_DIS
LIN {X -0.171,Y -499.785,Z 308.538,A 0.000,B 0.000,C 90.000,E1 96.891} C_DIS
LIN {X 0.185,Y -501.512,Z 308.537,A 0.000,B 0.000,C 90.000,E1 96.606} C_DIS
LIN {X 0.102,Y -502.807,Z 308.535,A 0.000,B 0.000,C 90.000,E1 96.372} C_DIS
LIN {X -0.105,Y -504.403,Z 308.533,A 0.000,B 0.000,C 90.000,E1 95.910} C_DIS
LIN {X 0.197,Y -504.914,Z 308.530,A 0.000,B 0.000,C 90.000,E1 95.391} C_DIS
LIN {X -0.040,Y -504.423,Z 308.527,A 0.000,B 0.000,C 90.000,E1 94.935} C_DIS
LIN {X -0.228,Y -502.847,Z 308.525,A 0.000,B 0.000,C 90.000,E1 94.473} C_DIS
LIN {X 0.157,Y -501.563,Z 308.523,A 0.000,B 0.000,C 90.000,E1 94.188} C_DIS
LIN {X -0.163,Y -496.190,Z 308.519,A 0.000,B 0.000,C 90.000,E1 93.498} C_DIS
LIN {X -0.174,Y -488.260,Z 308.514,A 0.000,B 0.000,C 90.000,E1 92.522} C_DIS
LIN {X 0.168,Y -473.669,Z 308.504,A 0.000,B 0.000,C 90.000,E1 90.745} C_DIS
LIN {X 0.005,Y -454.038,Z 308.490,A 0.000,B 0.000,C 90.000,E1 88.224} C_DIS
LIN {X -0.188,Y -436.356,Z 308.476,A 0.000,B 0.000,C 90.000,E1 85.641} C_DIS
LIN {X -0.079,Y -421.856,Z 308.462,A 0.000,B 0.000,C 90.000,E1 83.223} C_DIS
LIN {X 0.022,Y -404.297,Z 308.444,A 0.000,B 0.000,C 90.000,E1 79.926} C_DIS
LIN {X 0.174,Y -395.715,Z 308.435,A 0.000,B 0.000,C 90.000,E1 78.229} C_DIS
LIN {X -0.072,Y -385.537,Z 308.424,A 0.000,B 0.000,C 90.000,E1 76.284} C_DIS
LIN {X -0.149,Y -375.427,Z 308.413,A 0.000,B 0.000,C 90.000,E1 74.283} C_DIS
LIN {X -0.138,Y -365.345,Z 308.401,A 0.000,B 0.000,C 90.000,E1 72.236} C_DIS
LIN {X 0.057,Y -353.800,Z 308.388,A 0.000,B 0.000,C 90.000,E1 69.826} C_DIS
LIN {X 0.030,Y -338.390,Z 308.369,A 0.000,B 0.000,C 90.000,E1 66.485} C_DIS
LIN {X 0.060,Y -324.898,Z 308.350,A 0.000,B 0.000,C 90.000,E1 63.050} C_DIS
LIN {X -0.044,Y -314.587,Z 308.334,A 0.000,B 0.000,C 90.000,E1 60.205} C_DIS
LIN {X 0.098,Y -306.862,Z 308.322,A 0.000,B 0.000,C 90.000,E1 57.916} C_DIS
LIN {X 0.039,Y -297.435,Z 308.305,A 0.000,B 0.000,C 90.000,E1 54.975} C_DIS
LIN {X 0.013,Y -289.461,Z 308.291,A 0.000,B 0.000,C 90.000,E1 52.316} C_DIS
LIN {X -0.034,Y -281.606,Z 308.276,A 0.000,B 0.000,C 90.000,E1 49.622} C_DIS
LIN {X 0.043,Y -275.652,Z 308.264,A 0.000,B 0.000,C 90.000,E1 47.553} C_DIS
LIN {X -0.094,Y -266.093,Z 308.245,A 0.000,B 0.000,C 90.000,E1 44.109} C_DIS
LIN {X -0.119,Y -260.536,Z 308.233,A 0.000,B 0.000,C 90.000,E1 42.000} C_DIS
LIN {X -0.060,Y -254.854,Z 308.221,A 0.000,B 0.000,C 90.000,E1 39.850} C_DIS
LIN {X -0.039,Y -249.174,Z 308.209,A 0.000,B 0.000,C 90.000,E1 37.684} C_DIS
LIN {X -0.121,Y -243.312,Z 308.197,A 0.000,B 0.000,C 90.000,E1 35.518} C_DIS
LIN {X -0.046,Y -235.388,Z 308.181,A 0.000,B 0.000,C 90.000,E1 32.546} C_DIS
LIN {X -0.026,Y -227.771,Z 308.164,A 0.000,B 0.000,C 90.000,E1 29.539} C_DIS
LIN {X -0.021,Y -220.752,Z 308.147,A 0.000,B 0.000,C 90.000,E1 26.488} C_DIS
LIN {X 0.007,Y -214.457,Z 308.130,A 0.000,B 0.000,C 90.000,E1 23.387} C_DIS
LIN {X 0.023,Y -209.103,Z 308.113,A 0.000,B 0.000,C 90.000,E1 20.248} C_DIS
LIN {X -0.040,Y -204.414,Z 308.095,A 0.000,B 0.000,C 90.000,E1 17.094} C_DIS
LIN {X 0.042,Y -199.562,Z 308.073,A 0.000,B 0.000,C 90.000,E1 13.063} C_DIS
LIN {X -0.007,Y -195.717,Z 308.050,A 0.000,B 0.000,C 90.000,E1 9.029} C_DIS
LIN {X -0.066,Y -192.097,Z 308.018,A 0.000,B 0.000,C 90.000,E1 3.326} C_DIS
LIN {X -0.036,Y -192.785,Z 307.924,A 0.000,B 0.000,C 90.000,E1 346.353} C_DIS
LIN {X -0.098,Y -196.324,Z 307.897,A 0.000,B 0.000,C 90.000,E1 341.456} C_DIS
LIN {X 0.021,Y -200.363,Z 307.874,A 0.000,B 0.000,C 90.000,E1 337.358} C_DIS
LIN {X 0.023,Y -205.443,Z 307.852,A 0.000,B 0.000,C 90.000,E1 333.332} C_DIS
LIN {X 0.105,Y -211.564,Z 307.830,A 0.000,B 0.000,C 90.000,E1 329.331} C_DIS
LIN {X -0.008,Y -218.451,Z 307.808,A 0.000,B 0.000,C 90.000,E1 325.435} C_DIS
LIN {X -0.065,Y -224.708,Z 307.791,A 0.000,B 0.000,C 90.000,E1 322.351} C_DIS
LIN {X -0.090,Y -231.881,Z 307.774,A 0.000,B 0.000,C 90.000,E1 319.299} C_DIS
LIN {X -0.118,Y -240.163,Z 307.757,A 0.000,B 0.000,C 90.000,E1 316.296} C_DIS
LIN {X 0.072,Y -250.688,Z 307.739,A 0.000,B 0.000,C 90.000,E1 312.933} C_DIS
LIN {X -0.112,Y -262.241,Z 307.721,A 0.000,B 0.000,C 90.000,E1 309.725} C_DIS
LIN {X 0.110,Y -274.832,Z 307.703,A 0.000,B 0.000,C 90.000,E1 306.503} C_DIS
LIN {X 0.041,Y -288.783,Z 307.686,A 0.000,B 0.000,C 90.000,E1 303.420} C_DIS
LIN {X -0.031,Y -300.956,Z 307.673,A 0.000,B 0.000,C 90.000,E1 301.082} C_DIS
LIN {X 0.136,Y -318.116,Z 307.656,A 0.000,B 0.000,C 90.000,E1 298.103} C_DIS
LIN {X -0.078,Y -337.124,Z 307.640,A 0.000,B 0.000,C 90.000,E1 295.283} C_DIS
LIN {X -0.123,Y -352.540,Z 307.628,A 0.000,B 0.000,C 90.000,E1 293.131} C_DIS
LIN {X 0.154,Y -365.941,Z 307.618,A 0.000,B 0.000,C 90.000,E1 291.280} C_DIS
LIN {X -0.021,Y -386.469,Z 307.604,A 0.000,B 0.000,C 90.000,E1 288.671} C_DIS
LIN {X -0.079,Y -400.740,Z 307.594,A 0.000,B 0.000,C 90.000,E1 286.968} C_DIS
LIN {X -0.127,Y -414.904,Z 307.585,A 0.000,B 0.000,C 90.000,E1 285.300} C_DIS
LIN {X 0.232,Y -426.543,Z 307.577,A 0.000,B 0.000,C 90.000,E1 283.883} C_DIS
LIN {X -0.101,Y -433.113,Z 307.573,A 0.000,B 0.000,C 90.000,E1 283.119} C_DIS
LIN {X -0.186,Y -441.137,Z 307.567,A 0.000,B 0.000,C 90.000,E1 282.063} C_DIS
LIN {X -0.179,Y -448.594,Z 307.561,A 0.000,B 0.000,C 90.000,E1 281.007} C_DIS
LIN {X -0.170,Y -455.390,Z 307.555,A 0.000,B 0.000,C 90.000,E1 279.962} C_DIS
LIN {X -0.076,Y -461.680,Z 307.549,A 0.000,B 0.000,C 90.000,E1 278.916} C_DIS
LIN {X 0.168,Y -470.410,Z 307.541,A 0.000,B 0.000,C 90.000,E1 277.352} C_DIS
LIN {X -0.092,Y -475.834,Z 307.535,A 0.000,B 0.000,C 90.000,E1 276.372} C_DIS
LIN {X -0.156,Y -479.430,Z 307.531,A 0.000,B 0.000,C 90.000,E1 275.625} C_DIS
LIN {X -0.004,Y -481.498,Z 307.528,A 0.000,B 0.000,C 90.000,E1 275.106} C_DIS
LIN {X 0.161,Y -483.201,Z 307.526,A 0.000,B 0.000,C 90.000,E1 274.588} C_DIS
LIN {X -0.188,Y -484.536,Z 307.523,A 0.000,B 0.000,C 90.000,E1 274.131} C_DIS
LIN {X -0.009,Y -485.474,Z 307.520,A 0.000,B 0.000,C 90.000,E1 273.612} C_DIS
LIN {X 0.174,Y -486.040,Z 307.517,A 0.000,B 0.000,C 90.000,E1 273.094} C_DIS
LIN {X -0.149,Y -486.212,Z 307.515,A 0.000,B 0.000,C 90.000,E1 272.636} C_DIS
LIN {X 0.021,Y -486.099,Z 307.512,A 0.000,B 0.000,C 90.000,E1 272.121} C_DIS
LIN {X 0.206,Y -485.757,Z 307.509,A 0.000,B 0.000,C 90.000,E1 271.604} C_DIS
LIN {X 0.060,Y -484.623,Z 307.504,A 0.000,B 0.000,C 90.000,E1 270.630} C_DIS
LIN {X 0.226,Y -483.791,Z 307.501,A 0.000,B 0.000,C 90.000,E1 270.115} C_DIS
LIN {X -0.093,Y -482.611,Z 307.498,A 0.000,B 0.000,C 90.000,E1 269.656} C_DIS
LIN {X 0.064,Y -480.906,Z 307.495,A 0.000,B 0.000,C 90.000,E1 269.141} C_DIS
LIN {X 0.212,Y -478.596,Z 307.492,A 0.000,B 0.000,C 90.000,E1 268.625} C_DIS
LIN {X -0.120,Y -475.473,Z 307.490,A 0.000,B 0.000,C 90.000,E1 268.165} C_DIS
LIN {X 0.177,Y -473.591,Z 307.488,A 0.000,B 0.000,C 90.000,E1 267.879} C_DIS
LIN {X -0.002,Y -471.431,Z 307.487,A 0.000,B 0.000,C 90.000,E1 267.650} C_DIS
LIN {X 0.090,Y -466.130,Z 307.484,A 0.000,B 0.000,C 90.000,E1 267.135} C_DIS
LIN {X 0.053,Y -463.125,Z 307.483,A 0.000,B 0.000,C 90.000,E1 266.906} C_DIS
LIN {X 0.044,Y -459.708,Z 307.482,A 0.000,B 0.000,C 90.000,E1 266.674} C_DIS
LIN {X 0.182,Y -452.673,Z 307.479,A 0.000,B 0.000,C 90.000,E1 266.274} C_DIS
LIN {X 0.036,Y -445.113,Z 307.478,A 0.000,B 0.000,C 90.000,E1 265.988} C_DIS
LIN {X 0.064,Y -436.890,Z 307.476,A 0.000,B 0.000,C 90.000,E1 265.755} C_DIS
LIN {X -0.101,Y -432.701,Z 307.476,A 0.000,B 0.000,C 90.000,E1 265.698} C_DIS
LIN {X 0.164,Y -426.616,Z 307.476,A 0.000,B 0.000,C 90.000,E1 265.584} C_DIS
LIN {X 0.165,Y -418.414,Z 307.475,A 0.000,B 0.000,C 90.000,E1 265.527} C_DIS
LIN {X 0.036,Y -180.907,Z 307.475,A 0.000,B 0.000,C 90.000,E1 265.527} C_DIS
LIN {X 0.022,Y -180.756,Z 307.470,A 0.000,B 0.000,C 90.000,E1 264.666} C_DIS
LIN {X -0.086,Y -178.849,Z 307.442,A 0.000,B 0.000,C 90.000,E1 259.634} C_DIS
LIN {X -0.015,Y -175.893,Z 307.414,A 0.000,B 0.000,C 90.000,E1 254.519} C_DIS
LIN {X 0.091,Y -174.564,Z 307.405,A 0.000,B 0.000,C 90.000,E1 252.779} C_DIS
LIN {X -0.039,Y -171.549,Z 307.381,A 0.000,B 0.000,C 90.000,E1 248.539} C_DIS
LIN {X 0.016,Y -167.773,Z 307.357,A 0.000,B 0.000,C 90.000,E1 244.204} C_DIS
LIN {X -0.042,Y -166.483,Z 307.347,A 0.000,B 0.000,C 90.000,E1 242.487} C_DIS
LIN {X -0.046,Y -163.195,Z 307.328,A 0.000,B 0.000,C 90.000,E1 238.997} C_DIS
LIN {X 0.009,Y -161.158,Z 307.313,A 0.000,B 0.000,C 90.000,E1 236.342} C_DIS
LIN {X 0.044,Y -157.174,Z 307.288,A 0.000,B 0.000,C 90.000,E1 231.904} C_DIS
LIN {X -0.033,Y -155.905,Z 307.279,A 0.000,B 0.000,C 90.000,E1 230.150} C_DIS
LIN {X 0.024,Y -152.155,Z 307.254,A 0.000,B 0.000,C 90.000,E1 225.648} C_DIS
LIN {X 0.044,Y -150.405,Z 307.239,A 0.000,B 0.000,C 90.000,E1 222.933} C_DIS
LIN {X 0.067,Y -147.134,Z 307.213,A 0.000,B 0.000,C 90.000,E1 218.382} C_DIS
LIN {X -0.027,Y -145.696,Z 307.198,A 0.000,B 0.000,C 90.000,E1 215.678} C_DIS
LIN {X 0.055,Y -143.078,Z 307.173,A 0.000,B 0.000,C 90.000,E1 211.052} C_DIS
LIN {X -0.014,Y -141.696,Z 307.152,A 0.000,B 0.000,C 90.000,E1 207.385} C_DIS
LIN {X 0.040,Y -139.465,Z 307.116,A 0.000,B 0.000,C 90.000,E1 200.865} C_DIS
LIN {X -0.036,Y -139.198,Z 307.106,A 0.000,B 0.000,C 90.000,E1 199.033} C_DIS
LIN {X 0.026,Y -138.327,Z 307.054,A 0.000,B 0.000,C 90.000,E1 189.670} C_DIS
LIN {X 0.032,Y -139.447,Z 307.007,A 0.000,B 0.000,C 90.000,E1 181.260} C_DIS
LIN {X -0.028,Y -140.988,Z 306.976,A 0.000,B 0.000,C 90.000,E1 175.698} C_DIS
LIN {X 0.063,Y -142.742,Z 306.955,A 0.000,B 0.000,C 90.000,E1 171.951} C_DIS
LIN {X 0.019,Y -145.138,Z 306.930,A 0.000,B 0.000,C 90.000,E1 167.353} C_DIS
LIN {X 0.013,Y -147.761,Z 306.909,A 0.000,B 0.000,C 90.000,E1 163.685} C_DIS
LIN {X -0.048,Y -150.433,Z 306.889,A 0.000,B 0.000,C 90.000,E1 160.061} C_DIS
LIN {X -0.033,Y -153.877,Z 306.869,A 0.000,B 0.000,C 90.000,E1 156.433} C_DIS
LIN {X 0.022,Y -157.287,Z 306.849,A 0.000,B 0.000,C 90.000,E1 152.820} C_DIS
LIN {X -0.041,Y -161.469,Z 306.829,A 0.000,B 0.000,C 90.000,E1 149.282} C_DIS
LIN {X -0.034,Y -165.669,Z 306.810,A 0.000,B 0.000,C 90.000,E1 145.754} C_DIS
LIN {X -0.054,Y -170.607,Z 306.790,A 0.000,B 0.000,C 90.000,E1 142.271} C_DIS
LIN {X 0.100,Y -175.484,Z 306.771,A 0.000,B 0.000,C 90.000,E1 138.771} C_DIS
LIN {X -0.033,Y -181.105,Z 306.752,A 0.000,B 0.000,C 90.000,E1 135.405} C_DIS
LIN {X -0.043,Y -186.550,Z 306.733,A 0.000,B 0.000,C 90.000,E1 132.043} C_DIS
LIN {X -0.103,Y -191.165,Z 306.720,A 0.000,B 0.000,C 90.000,E1 129.564} C_DIS
LIN {X 0.092,Y -196.969,Z 306.701,A 0.000,B 0.000,C 90.000,E1 126.217} C_DIS
LIN {X 0.010,Y -200.236,Z 306.692,A 0.000,B 0.000,C 90.000,E1 124.612} C_DIS
LIN {X 0.121,Y -202.163,Z 306.686,A 0.000,B 0.000,C 90.000,E1 123.499} C_DIS
LIN {X 0.146,Y -303.332,Z 306.686,A 0.000,B 0.000,C 90.000,E1 123.499} C_DIS
LIN {X -0.116,Y -306.127,Z 306.686,A 0.000,B 0.000,C 90.000,E1 123.499} C_DIS
LIN {X -0.039,Y -310.642,Z 306.685,A 0.000,B 0.000,C 90.000,E1 123.245} C_DIS
LIN {X -0.052,Y -313.231,Z 306.683,A 0.000,B 0.000,C 90.000,E1 123.007} C_DIS
LIN {X 0.009,Y -316.982,Z 306.680,A 0.000,B 0.000,C 90.000,E1 122.467} C_DIS
LIN {X 0.069,Y -318.576,Z 306.679,A 0.000,B 0.000,C 90.000,E1 122.133} C_DIS
LIN {X 0.188,Y -332.115,Z 306.659,A 0.000,B 0.000,C 90.000,E1 118.615} C_DIS
LIN {X 0.010,Y -344.664,Z 306.644,A 0.000,B 0.000,C 90.000,E1 115.848} C_DIS
LIN {X 0.159,Y -357.103,Z 306.630,A 0.000,B 0.000,C 90.000,E1 113.387} C_DIS
LIN {X -0.130,Y -370.845,Z 306.617,A 0.000,B 0.000,C 90.000,E1 111.046} C_DIS
LIN {X 0.148,Y -385.989,Z 306.604,A 0.000,B 0.000,C 90.000,E1 108.671} C_DIS
LIN {X -0.179,Y -402.649,Z 306.591,A 0.000,B 0.000,C 90.000,E1 106.441} C_DIS
LIN {X 0.063,Y -420.948,Z 306.579,A 0.000,B 0.000,C 90.000,E1 104.189} C_DIS
LIN {X 0.044,Y -440.751,Z 306.567,A 0.000,B 0.000,C 90.000,E1 102.063} C_DIS
LIN {X -0.247,Y -461.217,Z 306.556,A 0.000,B 0.000,C 90.000,E1 100.141} C_DIS
LIN {X -0.056,Y -484.858,Z 306.545,A 0.000,B 0.000,C 90.000,E1 98.106} C_DIS
LIN {X -0.035,Y -498.030,Z 306.539,A 0.000,B 0.000,C 90.000,E1 97.068} C_DIS
LIN {X 0.249,Y -499.929,Z 306.538,A 0.000,B 0.000,C 90.000,E1 96.834} C_DIS
LIN {X 0.110,Y -501.678,Z 306.537,A 0.000,B 0.000,C 90.000,E1 96.606} C_DIS
LIN {X 0.026,Y -502.989,Z 306.535,A 0.000,B 0.000,C 90.000,E1 96.372} C_DIS
LIN {X -0.179,Y -504.611,Z 306.533,A 0.000,B 0.000,C 90.000,E1 95.910} C_DIS
LIN {X 0.123,Y -505.145,Z 306.530,A 0.000,B 0.000,C 90.000,E1 95.391} C_DIS
LIN {X -0.113,Y -504.678,Z 306.527,A 0.000,B 0.000,C 90.000,E1 94.935} C_DIS
LIN {X 0.201,Y -503.131,Z 306.525,A 0.000,B 0.000,C 90.000,E1 94.416} C_DIS
LIN {X 0.087,Y -501.864,Z 306.523,A 0.000,B 0.000,C 90.000,E1 94.188} C_DIS
LIN {X -0.231,Y -496.528,Z 306.519,A 0.000,B 0.000,C 90.000,E1 93.498} C_DIS
LIN {X -0.237,Y -488.587,Z 306.514,A 0.000,B 0.000,C 90.000,E1 92.522} C_DIS
LIN {X 0.113,Y -473.969,Z 306.504,A 0.000,B 0.000,C 90.000,E1 90.745} C_DIS
LIN {X -0.039,Y -454.283,Z 306.490,A 0.000,B 0.000,C 90.000,E1 88.224} C_DIS
LIN {X 0.212,Y -436.586,Z 306.476,A 0.000,B 0.000,C 90.000,E1 85.584} C_DIS
LIN {X -0.108,Y -422.069,Z 306.462,A 0.000,B 0.000,C 90.000,E1 83.223} C_DIS
LIN {X 0.002,Y -404.515,Z 306.444,A 0.000,B 0.000,C 90.000,E1 79.926} C_DIS
LIN {X 0.158,Y -395.932,Z 306.435,A 0.000,B 0.000,C 90.000,E1 78.229} C_DIS
LIN {X -0.084,Y -385.756,Z 306.424,A 0.000,B 0.000,C 90.000,E1 76.284} C_DIS
LIN {X -0.055,Y -375.652,Z 306.413,A 0.000,B 0.000,C 90.000,E1 74.267} C_DIS
LIN {X -0.139,Y -365.574,Z 306.401,A 0.000,B 0.000,C 90.000,E1 72.236} C_DIS
LIN {X 0.011,Y -355.495,Z 306.390,A 0.000,B 0.000,C 90.000,E1 70.134} C_DIS
LIN {X 0.012,Y -342.714,Z 306.375,A 0.000,B 0.000,C 90.000,E1 67.411} C_DIS
LIN {X -0.164,Y -332.347,Z 306.361,A 0.000,B 0.000,C 90.000,E1 64.973} C_DIS
LIN {X 0.167,Y -320.569,Z 306.343,A 0.000,B 0.000,C 90.000,E1 61.769} C_DIS
LIN {X 0.031,Y -309.387,Z 306.326,A 0.000,B 0.000,C 90.000,E1 58.584} C_DIS
LIN {X 0.081,Y -297.732,Z 306.306,A 0.000,B 0.000,C 90.000,E1 54.975} C_DIS
LIN {X -0.034,Y -291.741,Z 306.294,A 0.000,B 0.000,C 90.000,E1 53.004} C_DIS
LIN {X 0.087,Y -285.786,Z 306.283,A 0.000,B 0.000,C 90.000,E1 50.964} C_DIS
LIN {X 0.058,Y -279.869,Z 306.272,A 0.000,B 0.000,C 90.000,E1 48.933} C_DIS
LIN {X 0.056,Y -270.066,Z 306.253,A 0.000,B 0.000,C 90.000,E1 45.486} C_DIS
LIN {X 0.023,Y -262.606,Z 306.237,A 0.000,B 0.000,C 90.000,E1 42.690} C_DIS
LIN {X 0.121,Y -256.978,Z 306.225,A 0.000,B 0.000,C 90.000,E1 40.539} C_DIS
LIN {X 0.137,Y -251.290,Z 306.213,A 0.000,B 0.000,C 90.000,E1 38.382} C_DIS
LIN {X 0.087,Y -245.507,Z 306.201,A 0.000,B 0.000,C 90.000,E1 36.217} C_DIS
LIN {X -0.018,Y -239.537,Z 306.189,A 0.000,B 0.000,C 90.000,E1 34.040} C_DIS
LIN {X 0.025,Y -231.746,Z 306.173,A 0.000,B 0.000,C 90.000,E1 31.052} C_DIS
LIN {X 0.032,Y -224.364,Z 306.156,A 0.000,B 0.000,C 90.000,E1 28.025} C_DIS
LIN {X 0.044,Y -217.737,Z 306.139,A 0.000,B 0.000,C 90.000,E1 24.951} C_DIS
LIN {X 0.019,Y -211.944,Z 306.121,A 0.000,B 0.000,C 90.000,E1 21.844} C_DIS
LIN {X 0.111,Y -205.772,Z 306.099,A 0.000,B 0.000,C 90.000,E1 17.873} C_DIS
LIN {X 0.087,Y -200.673,Z 306.077,A 0.000,B 0.000,C 90.000,E1 13.883} C_DIS
LIN {X 0.071,Y -196.639,Z 306.055,A 0.000,B 0.000,C 90.000,E1 9.849} C_DIS
LIN {X -0.048,Y -193.202,Z 306.028,A 0.000,B 0.000,C 90.000,E1 4.992} C_DIS
LIN {X 0.084,Y -190.780,Z 305.993,A 0.000,B 0.000,C 90.000,E1 358.682} C_DIS
LIN {X -0.006,Y -192.111,Z 305.933,A 0.000,B 0.000,C 90.000,E1 347.993} C_DIS
LIN {X -0.063,Y -195.098,Z 305.906,A 0.000,B 0.000,C 90.000,E1 343.087} C_DIS
LIN {X -0.122,Y -198.750,Z 305.883,A 0.000,B 0.000,C 90.000,E1 339.028} C_DIS
LIN {X -0.073,Y -203.388,Z 305.861,A 0.000,B 0.000,C 90.000,E1 334.973} C_DIS
LIN {X 0.113,Y -209.110,Z 305.839,A 0.000,B 0.000,C 90.000,E1 330.923} C_DIS
LIN {X 0.052,Y -215.641,Z 305.817,A 0.000,B 0.000,C 90.000,E1 326.993} C_DIS
LIN {X -0.055,Y -223.165,Z 305.795,A 0.000,B 0.000,C 90.000,E1 323.130} C_DIS
LIN {X -0.086,Y -230.118,Z 305.778,A 0.000,B 0.000,C 90.000,E1 320.070} C_DIS
LIN {X 0.008,Y -238.140,Z 305.761,A 0.000,B 0.000,C 90.000,E1 317.025} C_DIS
LIN {X -0.041,Y -248.434,Z 305.743,A 0.000,B 0.000,C 90.000,E1 313.704} C_DIS
LIN {X -0.128,Y -259.756,Z 305.725,A 0.000,B 0.000,C 90.000,E1 310.458} C_DIS
LIN {X 0.017,Y -272.102,Z 305.707,A 0.000,B 0.000,C 90.000,E1 307.237} C_DIS
LIN {X 0.034,Y -285.704,Z 305.690,A 0.000,B 0.000,C 90.000,E1 304.119} C_DIS
LIN {X 0.050,Y -297.553,Z 305.676,A 0.000,B 0.000,C 90.000,E1 301.750} C_DIS
LIN {X -0.153,Y -314.413,Z 305.660,A 0.000,B 0.000,C 90.000,E1 298.821} C_DIS
LIN {X 0.063,Y -335.214,Z 305.642,A 0.000,B 0.000,C 90.000,E1 295.591} C_DIS
LIN {X -0.153,Y -350.555,Z 305.630,A 0.000,B 0.000,C 90.000,E1 293.462} C_DIS
LIN {X -0.111,Y -363.906,Z 305.620,A 0.000,B 0.000,C 90.000,E1 291.642} C_DIS
LIN {X -0.121,Y -379.599,Z 305.609,A 0.000,B 0.000,C 90.000,E1 289.577} C_DIS
LIN {X 0.115,Y -396.067,Z 305.597,A 0.000,B 0.000,C 90.000,E1 287.528} C_DIS
LIN {X -0.103,Y -409.994,Z 305.588,A 0.000,B 0.000,C 90.000,E1 285.898} C_DIS
LIN {X -0.086,Y -424.019,Z 305.579,A 0.000,B 0.000,C 90.000,E1 284.245} C_DIS
LIN {X 0.069,Y -430.716,Z 305.575,A 0.000,B 0.000,C 90.000,E1 283.411} C_DIS
LIN {X 0.194,Y -436.938,Z 305.570,A 0.000,B 0.000,C 90.000,E1 282.591} C_DIS
LIN {X 0.160,Y -444.641,Z 305.564,A 0.000,B 0.000,C 90.000,E1 281.535} C_DIS
LIN {X 0.128,Y -451.762,Z 305.558,A 0.000,B 0.000,C 90.000,E1 280.489} C_DIS
LIN {X 0.186,Y -458.287,Z 305.553,A 0.000,B 0.000,C 90.000,E1 279.443} C_DIS
LIN {X -0.137,Y -464.311,Z 305.547,A 0.000,B 0.000,C 90.000,E1 278.454} C_DIS
LIN {X -0.160,Y -471.500,Z 305.540,A 0.000,B 0.000,C 90.000,E1 277.182} C_DIS
LIN {X 0.065,Y -476.795,Z 305.534,A 0.000,B 0.000,C 90.000,E1 276.144} C_DIS
LIN {X 0.062,Y -480.228,Z 305.530,A 0.000,B 0.000,C 90.000,E1 275.391} C_DIS
LIN {X 0.038,Y -482.965,Z 305.526,A 0.000,B 0.000,C 90.000,E1 274.645} C_DIS
LIN {X 0.169,Y -484.350,Z 305.523,A 0.000,B 0.000,C 90.000,E1 274.131} C_DIS
LIN {X -0.137,Y -485.325,Z 305.520,A 0.000,B 0.000,C 90.000,E1 273.669} C_DIS
LIN {X 0.019,Y -485.921,Z 305.518,A 0.000,B 0.000,C 90.000,E1 273.154} C_DIS
LIN {X 0.207,Y -486.141,Z 305.515,A 0.000,B 0.000,C 90.000,E1 272.636} C_DIS
LIN {X -0.110,Y -486.048,Z 305.512,A 0.000,B 0.000,C 90.000,E1 272.178} C_DIS
LIN {X -0.240,Y -485.219,Z 305.507,A 0.000,B 0.000,C 90.000,E1 271.203} C_DIS
LIN {X -0.071,Y -484.652,Z 305.504,A 0.000,B 0.000,C 90.000,E1 270.688} C_DIS
LIN {X 0.095,Y -483.870,Z 305.501,A 0.000,B 0.000,C 90.000,E1 270.172} C_DIS
LIN {X -0.225,Y -482.686,Z 305.498,A 0.000,B 0.000,C 90.000,E1 269.714} C_DIS
LIN {X -0.066,Y -481.084,Z 305.496,A 0.000,B 0.000,C 90.000,E1 269.198} C_DIS
LIN {X 0.083,Y -478.864,Z 305.493,A 0.000,B 0.000,C 90.000,E1 268.682} C_DIS
LIN {X 0.214,Y -475.845,Z 305.490,A 0.000,B 0.000,C 90.000,E1 268.167} C_DIS
LIN {X -0.126,Y -471.889,Z 305.487,A 0.000,B 0.000,C 90.000,E1 267.707} C_DIS
LIN {X 0.157,Y -469.470,Z 305.486,A 0.000,B 0.000,C 90.000,E1 267.421} C_DIS
LIN {X -0.078,Y -463.856,Z 305.483,A 0.000,B 0.000,C 90.000,E1 266.963} C_DIS
LIN {X 0.195,Y -457.334,Z 305.481,A 0.000,B 0.000,C 90.000,E1 266.502} C_DIS
LIN {X 0.029,Y -453.783,Z 305.480,A 0.000,B 0.000,C 90.000,E1 266.331} C_DIS
LIN {X -0.223,Y -446.157,Z 305.478,A 0.000,B 0.000,C 90.000,E1 266.045} C_DIS
LIN {X 0.198,Y -442.543,Z 305.477,A 0.000,B 0.000,C 90.000,E1 265.869} C_DIS
LIN {X 0.146,Y -437.961,Z 305.477,A 0.000,B 0.000,C 90.000,E1 265.755} C_DIS
LIN {X 0.186,Y -428.439,Z 305.476,A 0.000,B 0.000,C 90.000,E1 265.584} C_DIS
LIN {X 0.010,Y -417.687,Z 305.475,A 0.000,B 0.000,C 90.000,E1 265.527} C_DIS
LIN {X -0.018,Y -180.908,Z 305.475,A 0.000,B 0.000,C 90.000,E1 265.527} C_DIS
LIN {X 0.014,Y -180.672,Z 305.469,A 0.000,B 0.000,C 90.000,E1 264.489} C_DIS
LIN {X 0.020,Y -179.017,Z 305.445,A 0.000,B 0.000,C 90.000,E1 260.095} C_DIS
LIN {X -0.061,Y -178.645,Z 305.440,A 0.000,B 0.000,C 90.000,E1 259.275} C_DIS
LIN {X 0.012,Y -175.696,Z 305.412,A 0.000,B 0.000,C 90.000,E1 254.157} C_DIS
LIN {X 0.024,Y -172.413,Z 305.388,A 0.000,B 0.000,C 90.000,E1 249.880} C_DIS
LIN {X 0.040,Y -171.228,Z 305.379,A 0.000,B 0.000,C 90.000,E1 248.156} C_DIS
LIN {X 0.015,Y -167.509,Z 305.355,A 0.000,B 0.000,C 90.000,E1 243.845} C_DIS
LIN {X -0.052,Y -166.905,Z 305.350,A 0.000,B 0.000,C 90.000,E1 242.999} C_DIS
LIN {X 0.001,Y -162.212,Z 305.321,A 0.000,B 0.000,C 90.000,E1 237.740} C_DIS
LIN {X -0.079,Y -160.790,Z 305.311,A 0.000,B 0.000,C 90.000,E1 236.008} C_DIS
LIN {X 0.025,Y -157.580,Z 305.291,A 0.000,B 0.000,C 90.000,E1 232.431} C_DIS
LIN {X 0.059,Y -155.613,Z 305.276,A 0.000,B 0.000,C 90.000,E1 229.747} C_DIS
LIN {X 0.002,Y -151.891,Z 305.252,A 0.000,B 0.000,C 90.000,E1 225.283} C_DIS
LIN {X -0.091,Y -150.120,Z 305.237,A 0.000,B 0.000,C 90.000,E1 222.609} C_DIS
LIN {X 0.038,Y -146.912,Z 305.211,A 0.000,B 0.000,C 90.000,E1 218.016} C_DIS
LIN {X -0.061,Y -145.499,Z 305.196,A 0.000,B 0.000,C 90.000,E1 215.311} C_DIS
LIN {X 0.057,Y -142.903,Z 305.171,A 0.000,B 0.000,C 90.000,E1 210.669} C_DIS
LIN {X -0.012,Y -141.524,Z 305.150,A 0.000,B 0.000,C 90.000,E1 207.001} C_DIS
LIN {X 0.031,Y -139.396,Z 305.114,A 0.000,B 0.000,C 90.000,E1 200.482} C_DIS
LIN {X 0.082,Y -139.108,Z 305.104,A 0.000,B 0.000,C 90.000,E1 198.598} C_DIS
LIN {X -0.062,Y -138.352,Z 305.057,A 0.000,B 0.000,C 90.000,E1 190.254} C_DIS
LIN {X 0.067,Y -139.510,Z 305.005,A 0.000,B 0.000,C 90.000,E1 180.859} C_DIS
LIN {X 0.008,Y -141.151,Z 304.974,A 0.000,B 0.000,C 90.000,E1 175.298} C_DIS
LIN {X -0.021,Y -142.531,Z 304.958,A 0.000,B 0.000,C 90.000,E1 172.527} C_DIS
LIN {X 0.047,Y -144.799,Z 304.933,A 0.000,B 0.000,C 90.000,E1 167.881} C_DIS
LIN {X 0.035,Y -147.418,Z 304.912,A 0.000,B 0.000,C 90.000,E1 164.212} C_DIS
LIN {X 0.064,Y -149.994,Z 304.892,A 0.000,B 0.000,C 90.000,E1 160.550} C_DIS
LIN {X 0.072,Y -153.323,Z 304.872,A 0.000,B 0.000,C 90.000,E1 156.922} C_DIS
LIN {X -0.017,Y -155.022,Z 304.862,A 0.000,B 0.000,C 90.000,E1 155.153} C_DIS
LIN {X 0.006,Y -158.670,Z 304.842,A 0.000,B 0.000,C 90.000,E1 151.563} C_DIS
LIN {X 0.088,Y -161.948,Z 304.827,A 0.000,B 0.000,C 90.000,E1 148.869} C_DIS
LIN {X -0.028,Y -166.139,Z 304.808,A 0.000,B 0.000,C 90.000,E1 145.388} C_DIS
LIN {X -0.032,Y -171.151,Z 304.788,A 0.000,B 0.000,C 90.000,E1 141.904} C_DIS
LIN {X 0.003,Y -176.029,Z 304.769,A 0.000,B 0.000,C 90.000,E1 138.447} C_DIS
LIN {X -0.001,Y -180.282,Z 304.755,A 0.000,B 0.000,C 90.000,E1 135.891} C_DIS
LIN {X -0.029,Y -185.694,Z 304.736,A 0.000,B 0.000,C 90.000,E1 132.528} C_DIS
LIN {X 0.024,Y -190.299,Z 304.722,A 0.000,B 0.000,C 90.000,E1 130.011} C_DIS
LIN {X 0.072,Y -197.625,Z 304.699,A 0.000,B 0.000,C 90.000,E1 125.884} C_DIS
LIN {X 0.042,Y -201.352,Z 304.689,A 0.000,B 0.000,C 90.000,E1 123.992} C_DIS
LIN {X 0.015,Y -202.216,Z 304.686,A 0.000,B 0.000,C 90.000,E1 123.499} C_DIS
LIN {X -0.023,Y -303.407,Z 304.686,A 0.000,B 0.000,C 90.000,E1 123.499} C_DIS
LIN {X 0.098,Y -305.300,Z 304.686,A 0.000,B 0.000,C 90.000,E1 123.452} C_DIS
LIN {X -0.146,Y -308.596,Z 304.685,A 0.000,B 0.000,C 90.000,E1 123.372} C_DIS
LIN {X 0.117,Y -311.902,Z 304.684,A 0.000,B 0.000,C 90.000,E1 123.086} C_DIS
LIN {X 0.034,Y -315.574,Z 304.682,A 0.000,B 0.000,C 90.000,E1 122.673} C_DIS
LIN {X 0.143,Y -317.460,Z 304.680,A 0.000,B 0.000,C 90.000,E1 122.339} C_DIS
LIN {X -0.018,Y -318.934,Z 304.678,A 0.000,B 0.000,C 90.000,E1 122.054} C_DIS
LIN {X -0.001,Y -331.163,Z 304.660,A 0.000,B 0.000,C 90.000,E1 118.871} C_DIS
LIN {X 0.095,Y -343.596,Z 304.645,A 0.000,B 0.000,C 90.000,E1 116.052} C_DIS
LIN {X -0.099,Y -355.924,Z 304.631,A 0.000,B 0.000,C 90.000,E1 113.643} C_DIS
LIN {X 0.056,Y -369.545,Z 304.618,A 0.000,B 0.000,C 90.000,E1 111.227} C_DIS
LIN {X -0.058,Y -384.561,Z 304.605,A 0.000,B 0.000,C 90.000,E1 108.906} C_DIS
LIN {X -0.048,Y -401.081,Z 304.592,A 0.000,B 0.000,C 90.000,E1 106.622} C_DIS
LIN {X -0.141,Y -419.228,Z 304.580,A 0.000,B 0.000,C 90.000,E1 104.411} C_DIS
LIN {X 0.055,Y -438.938,Z 304.568,A 0.000,B 0.000,C 90.000,E1 102.243} C_DIS
LIN {X 0.182,Y -459.356,Z 304.557,A 0.000,B 0.000,C 90.000,E1 100.254} C_DIS
LIN {X 0.261,Y -482.951,Z 304.546,A 0.000,B 0.000,C 90.000,E1 98.219} C_DIS
LIN {X 0.219,Y -496.285,Z 304.540,A 0.000,B 0.000,C 90.000,E1 97.182} C_DIS
LIN {X -0.003,Y -498.682,Z 304.539,A 0.000,B 0.000,C 90.000,E1 97.004} C_DIS
LIN {X 0.156,Y -502.107,Z 304.536,A 0.000,B 0.000,C 90.000,E1 96.549} C_DIS
LIN {X 0.074,Y -503.372,Z 304.535,A 0.000,B 0.000,C 90.000,E1 96.315} C_DIS
LIN {X -0.062,Y -504.298,Z 304.534,A 0.000,B 0.000,C 90.000,E1 96.087} C_DIS
LIN {X -0.258,Y -505.287,Z 304.531,A 0.000,B 0.000,C 90.000,E1 95.625} C_DIS
LIN {X 0.054,Y -505.256,Z 304.528,A 0.000,B 0.000,C 90.000,E1 95.106} C_DIS
LIN {X -0.133,Y -504.200,Z 304.526,A 0.000,B 0.000,C 90.000,E1 94.645} C_DIS
LIN {X -0.247,Y -503.235,Z 304.524,A 0.000,B 0.000,C 90.000,E1 94.416} C_DIS
LIN {X 0.142,Y -501.918,Z 304.523,A 0.000,B 0.000,C 90.000,E1 94.131} C_DIS
LIN {X -0.181,Y -496.527,Z 304.519,A 0.000,B 0.000,C 90.000,E1 93.440} C_DIS
LIN {X 0.159,Y -486.482,Z 304.512,A 0.000,B 0.000,C 90.000,E1 92.178} C_DIS
LIN {X -0.045,Y -461.864,Z 304.496,A 0.000,B 0.000,C 90.000,E1 89.198} C_DIS
LIN {X -0.014,Y -446.913,Z 304.484,A 0.000,B 0.000,C 90.000,E1 87.135} C_DIS
LIN {X 0.201,Y -428.285,Z 304.468,A 0.000,B 0.000,C 90.000,E1 84.204} C_DIS
LIN {X -0.144,Y -413.033,Z 304.453,A 0.000,B 0.000,C 90.000,E1 81.546} C_DIS
LIN {X -0.167,Y -401.648,Z 304.441,A 0.000,B 0.000,C 90.000,E1 79.342} C_DIS
LIN {X -0.059,Y -392.955,Z 304.431,A 0.000,B 0.000,C 90.000,E1 77.645} C_DIS
LIN {X 0.019,Y -382.818,Z 304.420,A 0.000,B 0.000,C 90.000,E1 75.644} C_DIS
LIN {X 0.073,Y -371.337,Z 304.407,A 0.000,B 0.000,C 90.000,E1 73.323} C_DIS
LIN {X -0.004,Y -361.241,Z 304.396,A 0.000,B 0.000,C 90.000,E1 71.275} C_DIS
LIN {X -0.128,Y -349.781,Z 304.383,A 0.000,B 0.000,C 90.000,E1 68.901} C_DIS
LIN {X 0.179,Y -337.441,Z 304.367,A 0.000,B 0.000,C 90.000,E1 66.102} C_DIS
LIN {X 0.128,Y -322.959,Z 304.347,A 0.000,B 0.000,C 90.000,E1 62.359} C_DIS
LIN {X -0.098,Y -311.687,Z 304.329,A 0.000,B 0.000,C 90.000,E1 59.203} C_DIS
LIN {X 0.002,Y -300.928,Z 304.311,A 0.000,B 0.000,C 90.000,E1 55.928} C_DIS
LIN {X -0.047,Y -292.851,Z 304.296,A 0.000,B 0.000,C 90.000,E1 53.290} C_DIS
LIN {X -0.015,Y -284.894,Z 304.281,A 0.000,B 0.000,C 90.000,E1 50.598} C_DIS
LIN {X -0.060,Y -278.938,Z 304.270,A 0.000,B 0.000,C 90.000,E1 48.566} C_DIS
LIN {X 0.097,Y -269.180,Z 304.251,A 0.000,B 0.000,C 90.000,E1 45.081} C_DIS
LIN {X 0.038,Y -261.751,Z 304.235,A 0.000,B 0.000,C 90.000,E1 42.285} C_DIS
LIN {X -0.050,Y -256.093,Z 304.223,A 0.000,B 0.000,C 90.000,E1 40.172} C_DIS
LIN {X -0.047,Y -250.408,Z 304.211,A 0.000,B 0.000,C 90.000,E1 38.016} C_DIS
LIN {X 0.088,Y -244.574,Z 304.199,A 0.000,B 0.000,C 90.000,E1 35.804} C_DIS
LIN {X -0.033,Y -238.595,Z 304.187,A 0.000,B 0.000,C 90.000,E1 33.627} C_DIS
LIN {X 0.039,Y -228.972,Z 304.166,A 0.000,B 0.000,C 90.000,E1 29.873} C_DIS
LIN {X -0.124,Y -221.889,Z 304.149,A 0.000,B 0.000,C 90.000,E1 26.873} C_DIS
LIN {X -0.063,Y -215.569,Z 304.132,A 0.000,B 0.000,C 90.000,E1 23.770} C_DIS
LIN {X 0.061,Y -210.132,Z 304.115,A 0.000,B 0.000,C 90.000,E1 20.610} C_DIS
LIN {X 0.022,Y -205.364,Z 304.097,A 0.000,B 0.000,C 90.000,E1 17.457} C_DIS
LIN {X -0.012,Y -200.387,Z 304.075,A 0.000,B 0.000,C 90.000,E1 13.467} C_DIS
LIN {X -0.042,Y -196.471,Z 304.052,A 0.000,B 0.000,C 90.000,E1 9.434} C_DIS
LIN {X -0.054,Y -192.705,Z 304.021,A 0.000,B 0.000,C 90.000,E1 3.726} C_DIS
LIN {X -0.001,Y -190.600,Z 303.975,A 0.000,B 0.000,C 90.000,E1 355.412} C_DIS
LIN {X 0.004,Y -192.654,Z 303.929,A 0.000,B 0.000,C 90.000,E1 347.173} C_DIS
LIN {X 0.075,Y -195.876,Z 303.901,A 0.000,B 0.000,C 90.000,E1 342.236} C_DIS
LIN {X 0.118,Y -199.713,Z 303.879,A 0.000,B 0.000,C 90.000,E1 338.156} C_DIS
LIN {X 0.020,Y -204.540,Z 303.856,A 0.000,B 0.000,C 90.000,E1 334.152} C_DIS
LIN {X -0.129,Y -210.440,Z 303.834,A 0.000,B 0.000,C 90.000,E1 330.205} C_DIS
LIN {X 0.076,Y -217.147,Z 303.812,A 0.000,B 0.000,C 90.000,E1 326.215} C_DIS
LIN {X -0.011,Y -223.275,Z 303.795,A 0.000,B 0.000,C 90.000,E1 323.130} C_DIS
LIN {X -0.039,Y -230.257,Z 303.778,A 0.000,B 0.000,C 90.000,E1 320.070} C_DIS
LIN {X -0.114,Y -238.318,Z 303.761,A 0.000,B 0.000,C 90.000,E1 317.067} C_DIS
LIN {X 0.018,Y -248.625,Z 303.743,A 0.000,B 0.000,C 90.000,E1 313.704} C_DIS
LIN {X -0.060,Y -259.933,Z 303.725,A 0.000,B 0.000,C 90.000,E1 310.458} C_DIS
LIN {X 0.094,Y -272.280,Z 303.707,A 0.000,B 0.000,C 90.000,E1 307.237} C_DIS
LIN {X 0.120,Y -285.894,Z 303.690,A 0.000,B 0.000,C 90.000,E1 304.119} C_DIS
LIN {X -0.110,Y -297.746,Z 303.677,A 0.000,B 0.000,C 90.000,E1 301.799} C_DIS
LIN {X -0.048,Y -314.684,Z 303.660,A 0.000,B 0.000,C 90.000,E1 298.821} C_DIS
LIN {X 0.184,Y -335.460,Z 303.642,A 0.000,B 0.000,C 90.000,E1 295.591} C_DIS
LIN {X -0.021,Y -350.812,Z 303.630,A 0.000,B 0.000,C 90.000,E1 293.462} C_DIS
LIN {X -0.042,Y -366.344,Z 303.619,A 0.000,B 0.000,C 90.000,E1 291.354} C_DIS
LIN {X 0.051,Y -389.103,Z 303.602,A 0.000,B 0.000,C 90.000,E1 288.417} C_DIS
LIN {X 0.054,Y -403.045,Z 303.593,A 0.000,B 0.000,C 90.000,E1 286.732} C_DIS
LIN {X 0.057,Y -417.051,Z 303.584,A 0.000,B 0.000,C 90.000,E1 285.064} C_DIS
LIN {X -0.216,Y -426.297,Z 303.578,A 0.000,B 0.000,C 90.000,E1 284.008} C_DIS
LIN {X -0.036,Y -432.800,Z 303.573,A 0.000,B 0.000,C 90.000,E1 283.175} C_DIS
LIN {X -0.125,Y -440.791,Z 303.567,A 0.000,B 0.000,C 90.000,E1 282.119} C_DIS
LIN {X -0.209,Y -448.154,Z 303.561,A 0.000,B 0.000,C 90.000,E1 281.074} C_DIS
LIN {X 0.072,Y -453.302,Z 303.557,A 0.000,B 0.000,C 90.000,E1 280.254} C_DIS
LIN {X 0.145,Y -459.690,Z 303.551,A 0.000,B 0.000,C 90.000,E1 279.208} C_DIS
LIN {X 0.064,Y -467.056,Z 303.544,A 0.000,B 0.000,C 90.000,E1 277.936} C_DIS
LIN {X -0.171,Y -472.697,Z 303.538,A 0.000,B 0.000,C 90.000,E1 276.947} C_DIS
LIN {X 0.063,Y -477.825,Z 303.533,A 0.000,B 0.000,C 90.000,E1 275.910} C_DIS
LIN {X 0.018,Y -481.052,Z 303.529,A 0.000,B 0.000,C 90.000,E1 275.163} C_DIS
LIN {X 0.180,Y -482.816,Z 303.526,A 0.000,B 0.000,C 90.000,E1 274.645} C_DIS
LIN {X -0.172,Y -484.221,Z 303.523,A 0.000,B 0.000,C 90.000,E1 274.188} C_DIS
LIN {X 0.004,Y -485.209,Z 303.520,A 0.000,B 0.000,C 90.000,E1 273.669} C_DIS
LIN {X 0.158,Y -485.815,Z 303.518,A 0.000,B 0.000,C 90.000,E1 273.154} C_DIS
LIN {X -0.139,Y -486.080,Z 303.515,A 0.000,B 0.000,C 90.000,E1 272.694} C_DIS
LIN {X 0.028,Y -485.986,Z 303.512,A 0.000,B 0.000,C 90.000,E1 272.178} C_DIS
LIN {X -0.103,Y -485.184,Z 303.507,A 0.000,B 0.000,C 90.000,E1 271.203} C_DIS
LIN {X 0.232,Y -483.896,Z 303.501,A 0.000,B 0.000,C 90.000,E1 270.172} C_DIS
LIN {X -0.088,Y -482.738,Z 303.498,A 0.000,B 0.000,C 90.000,E1 269.714} C_DIS
LIN {X 0.070,Y -481.168,Z 303.496,A 0.000,B 0.000,C 90.000,E1 269.198} C_DIS
LIN {X 0.219,Y -478.974,Z 303.493,A 0.000,B 0.000,C 90.000,E1 268.682} C_DIS
LIN {X 0.046,Y -477.618,Z 303.491,A 0.000,B 0.000,C 90.000,E1 268.453} C_DIS
LIN {X 0.187,Y -474.191,Z 303.489,A 0.000,B 0.000,C 90.000,E1 267.936} C_DIS
LIN {X -0.177,Y -469.713,Z 303.486,A 0.000,B 0.000,C 90.000,E1 267.478} C_DIS
LIN {X 0.051,Y -464.169,Z 303.483,A 0.000,B 0.000,C 90.000,E1 266.963} C_DIS
LIN {X 0.023,Y -460.881,Z 303.482,A 0.000,B 0.000,C 90.000,E1 266.731} C_DIS
LIN {X -0.190,Y -457.683,Z 303.481,A 0.000,B 0.000,C 90.000,E1 266.560} C_DIS
LIN {X 0.162,Y -450.583,Z 303.479,A 0.000,B 0.000,C 90.000,E1 266.159} C_DIS
LIN {X -0.205,Y -443.105,Z 303.477,A 0.000,B 0.000,C 90.000,E1 265.927} C_DIS
LIN {X 0.173,Y -438.657,Z 303.477,A 0.000,B 0.000,C 90.000,E1 265.755} C_DIS
LIN {X 0.166,Y -429.454,Z 303.476,A 0.000,B 0.000,C 90.000,E1 265.584} C_DIS
LIN {X 0.016,Y -421.746,Z 303.475,A 0.000,B 0.000,C 90.000,E1 265.527} C_DIS
LIN {X -0.102,Y -418.460,Z 303.475,A 0.000,B 0.000,C 90.000,E1 265.527} C_DIS
LIN {X -0.069,Y -180.907,Z 303.475,A 0.000,B 0.000,C 90.000,E1 265.527} C_DIS
LIN {X -0.017,Y -180.667,Z 303.469,A 0.000,B 0.000,C 90.000,E1 264.489} C_DIS
LIN {X -0.011,Y -179.014,Z 303.445,A 0.000,B 0.000,C 90.000,E1 260.095} C_DIS
LIN {X 0.084,Y -178.639,Z 303.440,A 0.000,B 0.000,C 90.000,E1 259.218} C_DIS
LIN {X -0.019,Y -175.689,Z 303.412,A 0.000,B 0.000,C 90.000,E1 254.157} C_DIS
LIN {X -0.007,Y -172.406,Z 303.388,A 0.000,B 0.000,C 90.000,E1 249.880} C_DIS
LIN {X 0.009,Y -171.218,Z 303.379,A 0.000,B 0.000,C 90.000,E1 248.156} C_DIS
LIN {X -0.015,Y -167.501,Z 303.355,A 0.000,B 0.000,C 90.000,E1 243.845} C_DIS
LIN {X -0.081,Y -166.898,Z 303.350,A 0.000,B 0.000,C 90.000,E1 242.999} C_DIS
LIN {X -0.029,Y -162.204,Z 303.321,A 0.000,B 0.000,C 90.000,E1 237.740} C_DIS
LIN {X 0.024,Y -160.779,Z 303.311,A 0.000,B 0.000,C 90.000,E1 235.960} C_DIS
LIN {X -0.004,Y -157.572,Z 303.291,A 0.000,B 0.000,C 90.000,E1 232.431} C_DIS
LIN {X 0.030,Y -155.603,Z 303.276,A 0.000,B 0.000,C 90.000,E1 229.747} C_DIS
LIN {X 0.080,Y -151.883,Z 303.252,A 0.000,B 0.000,C 90.000,E1 225.243} C_DIS
LIN {X 0.093,Y -150.110,Z 303.236,A 0.000,B 0.000,C 90.000,E1 222.528} C_DIS
LIN {X 0.010,Y -146.906,Z 303.211,A 0.000,B 0.000,C 90.000,E1 218.016} C_DIS
LIN {X -0.089,Y -145.493,Z 303.196,A 0.000,B 0.000,C 90.000,E1 215.311} C_DIS
LIN {X 0.030,Y -142.899,Z 303.170,A 0.000,B 0.000,C 90.000,E1 210.669} C_DIS
LIN {X -0.039,Y -141.520,Z 303.150,A 0.000,B 0.000,C 90.000,E1 207.001} C_DIS
LIN {X 0.004,Y -139.395,Z 303.114,A 0.000,B 0.000,C 90.000,E1 200.482} C_DIS
LIN {X 0.054,Y -139.106,Z 303.103,A 0.000,B 0.000,C 90.000,E1 198.598} C_DIS
LIN {X 0.047,Y -138.353,Z 303.057,A 0.000,B 0.000,C 90.000,E1 190.197} C_DIS
LIN {X 0.040,Y -139.511,Z 303.005,A 0.000,B 0.000,C 90.000,E1 180.859} C_DIS
LIN {X -0.019,Y -141.157,Z 302.974,A 0.000,B 0.000,C 90.000,E1 175.298} C_DIS
LIN {X -0.048,Y -142.536,Z 302.958,A 0.000,B 0.000,C 90.000,E1 172.527} C_DIS
LIN {X 0.020,Y -144.806,Z 302.933,A 0.000,B 0.000,C 90.000,E1 167.881} C_DIS
LIN {X 0.008,Y -147.426,Z 302.912,A 0.000,B 0.000,C 90.000,E1 164.212} C_DIS
LIN {X 0.036,Y -150.003,Z 302.892,A 0.000,B 0.000,C 90.000,E1 160.550} C_DIS
LIN {X 0.044,Y -153.334,Z 302.872,A 0.000,B 0.000,C 90.000,E1 156.922} C_DIS
LIN {X 0.025,Y -155.869,Z 302.857,A 0.000,B 0.000,C 90.000,E1 154.229} C_DIS
LIN {X -0.008,Y -159.722,Z 302.837,A 0.000,B 0.000,C 90.000,E1 150.667} C_DIS
LIN {X 0.058,Y -161.961,Z 302.827,A 0.000,B 0.000,C 90.000,E1 148.869} C_DIS
LIN {X -0.057,Y -166.152,Z 302.808,A 0.000,B 0.000,C 90.000,E1 145.388} C_DIS
LIN {X -0.062,Y -171.166,Z 302.788,A 0.000,B 0.000,C 90.000,E1 141.904} C_DIS
LIN {X -0.028,Y -176.045,Z 302.769,A 0.000,B 0.000,C 90.000,E1 138.447} C_DIS
LIN {X -0.032,Y -180.300,Z 302.755,A 0.000,B 0.000,C 90.000,E1 135.891} C_DIS
LIN {X -0.060,Y -185.711,Z 302.736,A 0.000,B 0.000,C 90.000,E1 132.528} C_DIS
LIN {X -0.009,Y -190.318,Z 302.722,A 0.000,B 0.000,C 90.000,E1 130.011} C_DIS
LIN {X 0.039,Y -197.644,Z 302.699,A 0.000,B 0.000,C 90.000,E1 125.884} C_DIS
LIN {X 0.000,Y -201.373,Z 302.689,A 0.000,B 0.000,C 90.000,E1 123.992} C_DIS
LIN {X 0.056,Y -202.279,Z 302.686,A 0.000,B 0.000,C 90.000,E1 123.452} C_DIS
LIN {X 0.046,Y -303.867,Z 302.686,A 0.000,B 0.000,C 90.000,E1 123.452} C_DIS
LIN {X -0.065,Y -307.723,Z 302.685,A 0.000,B 0.000,C 90.000,E1 123.372} C_DIS
LIN {X 0.059,Y -310.784,Z 302.684,A 0.000,B 0.000,C 90.000,E1 123.166} C_DIS
LIN {X -0.113,Y -314.458,Z 302.682,A 0.000,B 0.000,C 90.000,E1 122.832} C_DIS
LIN {X -0.047,Y -317.967,Z 302.679,A 0.000,B 0.000,C 90.000,E1 122.260} C_DIS
LIN {X 0.017,Y -319.386,Z 302.677,A 0.000,B 0.000,C 90.000,E1 121.926} C_DIS
LIN {X -0.066,Y -330.341,Z 302.661,A 0.000,B 0.000,C 90.000,E1 119.077} C_DIS
LIN {X 0.159,Y -342.673,Z 302.646,A 0.000,B 0.000,C 90.000,E1 116.232} C_DIS
LIN {X -0.060,Y -354.905,Z 302.632,A 0.000,B 0.000,C 90.000,E1 113.823} C_DIS
LIN {X 0.065,Y -368.423,Z 302.619,A 0.000,B 0.000,C 90.000,E1 111.408} C_DIS
LIN {X -0.078,Y -383.326,Z 302.606,A 0.000,B 0.000,C 90.000,E1 109.087} C_DIS
LIN {X -0.101,Y -399.727,Z 302.593,A 0.000,B 0.000,C 90.000,E1 106.804} C_DIS
LIN {X 0.178,Y -417.744,Z 302.581,A 0.000,B 0.000,C 90.000,E1 104.537} C_DIS
LIN {X -0.016,Y -437.368,Z 302.569,A 0.000,B 0.000,C 90.000,E1 102.411} C_DIS
LIN {X -0.008,Y -457.742,Z 302.558,A 0.000,B 0.000,C 90.000,E1 100.423} C_DIS
LIN {X -0.134,Y -481.297,Z 302.547,A 0.000,B 0.000,C 90.000,E1 98.398} C_DIS
LIN {X 0.021,Y -497.299,Z 302.540,A 0.000,B 0.000,C 90.000,E1 97.125} C_DIS
LIN {X 0.006,Y -501.196,Z 302.537,A 0.000,B 0.000,C 90.000,E1 96.720} C_DIS
LIN {X -0.079,Y -502.752,Z 302.536,A 0.000,B 0.000,C 90.000,E1 96.486} C_DIS
LIN {X -0.222,Y -503.913,Z 302.535,A 0.000,B 0.000,C 90.000,E1 96.258} C_DIS
LIN {X 0.081,Y -505.300,Z 302.532,A 0.000,B 0.000,C 90.000,E1 95.739} C_DIS
LIN {X -0.113,Y -505.631,Z 302.529,A 0.000,B 0.000,C 90.000,E1 95.277} C_DIS
LIN {X 0.202,Y -504.957,Z 302.527,A 0.000,B 0.000,C 90.000,E1 94.759} C_DIS
LIN {X -0.025,Y -503.155,Z 302.524,A 0.000,B 0.000,C 90.000,E1 94.302} C_DIS
LIN {X -0.137,Y -501.721,Z 302.523,A 0.000,B 0.000,C 90.000,E1 94.073} C_DIS
LIN {X 0.043,Y -496.220,Z 302.518,A 0.000,B 0.000,C 90.000,E1 93.326} C_DIS
LIN {X 0.030,Y -488.180,Z 302.513,A 0.000,B 0.000,C 90.000,E1 92.350} C_DIS
LIN {X 0.188,Y -471.461,Z 302.502,A 0.000,B 0.000,C 90.000,E1 90.344} C_DIS
LIN {X 0.204,Y -453.852,Z 302.489,A 0.000,B 0.000,C 90.000,E1 88.051} C_DIS
LIN {X -0.184,Y -437.900,Z 302.476,A 0.000,B 0.000,C 90.000,E1 85.755} C_DIS
LIN {X 0.075,Y -421.712,Z 302.461,A 0.000,B 0.000,C 90.000,E1 83.053} C_DIS
LIN {X -0.172,Y -404.215,Z 302.443,A 0.000,B 0.000,C 90.000,E1 79.803} C_DIS
LIN {X -0.091,Y -395.604,Z 302.434,A 0.000,B 0.000,C 90.000,E1 78.117} C_DIS
LIN {X 0.035,Y -385.461,Z 302.423,A 0.000,B 0.000,C 90.000,E1 76.117} C_DIS
LIN {X 0.153,Y -373.966,Z 302.410,A 0.000,B 0.000,C 90.000,E1 73.795} C_DIS
LIN {X 0.025,Y -363.887,Z 302.399,A 0.000,B 0.000,C 90.000,E1 71.764} C_DIS
LIN {X -0.040,Y -352.420,Z 302.385,A 0.000,B 0.000,C 90.000,E1 69.390} C_DIS
LIN {X -0.105,Y -337.320,Z 302.367,A 0.000,B 0.000,C 90.000,E1 66.049} C_DIS
LIN {X -0.007,Y -322.876,Z 302.346,A 0.000,B 0.000,C 90.000,E1 62.281} C_DIS
LIN {X 0.044,Y -311.624,Z 302.328,A 0.000,B 0.000,C 90.000,E1 59.076} C_DIS
LIN {X -0.092,Y -299.863,Z 302.308,A 0.000,B 0.000,C 90.000,E1 55.515} C_DIS
LIN {X 0.007,Y -291.816,Z 302.294,A 0.000,B 0.000,C 90.000,E1 52.844} C_DIS
LIN {X 0.014,Y -283.830,Z 302.279,A 0.000,B 0.000,C 90.000,E1 50.150} C_DIS
LIN {X 0.148,Y -275.837,Z 302.263,A 0.000,B 0.000,C 90.000,E1 47.391} C_DIS
LIN {X 0.014,Y -266.258,Z 302.244,A 0.000,B 0.000,C 90.000,E1 43.947} C_DIS
LIN {X -0.012,Y -260.710,Z 302.232,A 0.000,B 0.000,C 90.000,E1 41.838} C_DIS
LIN {X -0.116,Y -255.048,Z 302.221,A 0.000,B 0.000,C 90.000,E1 39.725} C_DIS
LIN {X 0.066,Y -249.344,Z 302.209,A 0.000,B 0.000,C 90.000,E1 37.523} C_DIS
LIN {X -0.021,Y -243.489,Z 302.196,A 0.000,B 0.000,C 90.000,E1 35.358} C_DIS
LIN {X -0.077,Y -235.530,Z 302.180,A 0.000,B 0.000,C 90.000,E1 32.418} C_DIS
LIN {X 0.100,Y -226.175,Z 302.159,A 0.000,B 0.000,C 90.000,E1 28.615} C_DIS
LIN {X -0.040,Y -219.414,Z 302.142,A 0.000,B 0.000,C 90.000,E1 25.591} C_DIS
LIN {X 0.064,Y -213.447,Z 302.125,A 0.000,B 0.000,C 90.000,E1 22.461} C_DIS
LIN {X 0.009,Y -207.129,Z 302.103,A 0.000,B 0.000,C 90.000,E1 18.544} C_DIS
LIN {X 0.088,Y -201.850,Z 302.081,A 0.000,B 0.000,C 90.000,E1 14.537} C_DIS
LIN {X -0.045,Y -197.674,Z 302.059,A 0.000,B 0.000,C 90.000,E1 10.546} C_DIS
LIN {X 0.091,Y -194.017,Z 302.031,A 0.000,B 0.000,C 90.000,E1 5.625} C_DIS
LIN {X -0.035,Y -191.359,Z 301.997,A 0.000,B 0.000,C 90.000,E1 359.542} C_DIS
LIN {X 0.022,Y -192.829,Z 301.929,A 0.000,B 0.000,C 90.000,E1 347.173} C_DIS
LIN {X 0.099,Y -196.014,Z 301.901,A 0.000,B 0.000,C 90.000,E1 342.236} C_DIS
LIN {X -0.040,Y -199.839,Z 301.879,A 0.000,B 0.000,C 90.000,E1 338.209} C_DIS
LIN {X 0.052,Y -204.659,Z 301.856,A 0.000,B 0.000,C 90.000,E1 334.152} C_DIS
LIN {X -0.092,Y -210.531,Z 301.834,A 0.000,B 0.000,C 90.000,E1 330.205} C_DIS
LIN {X 0.117,Y -217.233,Z 301.812,A 0.000,B 0.000,C 90.000,E1 326.215} C_DIS
LIN {X 0.033,Y -223.394,Z 301.795,A 0.000,B 0.000,C 90.000,E1 323.130} C_DIS
LIN {X 0.010,Y -230.400,Z 301.778,A 0.000,B 0.000,C 90.000,E1 320.070} C_DIS
LIN {X -0.053,Y -238.489,Z 301.761,A 0.000,B 0.000,C 90.000,E1 317.067} C_DIS
LIN {X 0.088,Y -248.810,Z 301.743,A 0.000,B 0.000,C 90.000,E1 313.704} C_DIS
LIN {X 0.017,Y -260.107,Z 301.725,A 0.000,B 0.000,C 90.000,E1 310.458} C_DIS
LIN {X -0.038,Y -272.451,Z 301.707,A 0.000,B 0.000,C 90.000,E1 307.282} C_DIS
LIN {X -0.183,Y -286.089,Z 301.690,A 0.000,B 0.000,C 90.000,E1 304.199} C_DIS
LIN {X -0.007,Y -297.963,Z 301.677,A 0.000,B 0.000,C 90.000,E1 301.799} C_DIS
LIN {X 0.067,Y -314.945,Z 301.660,A 0.000,B 0.000,C 90.000,E1 298.821} C_DIS
LIN {X -0.133,Y -335.697,Z 301.642,A 0.000,B 0.000,C 90.000,E1 295.668} C_DIS
LIN {X 0.120,Y -351.053,Z 301.630,A 0.000,B 0.000,C 90.000,E1 293.462} C_DIS
LIN {X 0.112,Y -366.531,Z 301.619,A 0.000,B 0.000,C 90.000,E1 291.354} C_DIS
LIN {X 0.219,Y -389.187,Z 301.603,A 0.000,B 0.000,C 90.000,E1 288.417} C_DIS
LIN {X 0.093,Y -403.216,Z 301.593,A 0.000,B 0.000,C 90.000,E1 286.732} C_DIS
LIN {X 0.098,Y -417.165,Z 301.584,A 0.000,B 0.000,C 90.000,E1 285.064} C_DIS
LIN {X -0.172,Y -426.369,Z 301.578,A 0.000,B 0.000,C 90.000,E1 284.008} C_DIS
LIN {X 0.010,Y -432.869,Z 301.573,A 0.000,B 0.000,C 90.000,E1 283.175} C_DIS
LIN {X -0.078,Y -440.763,Z 301.567,A 0.000,B 0.000,C 90.000,E1 282.119} C_DIS
LIN {X -0.161,Y -448.107,Z 301.561,A 0.000,B 0.000,C 90.000,E1 281.074} C_DIS
LIN {X -0.071,Y -454.867,Z 301.556,A 0.000,B 0.000,C 90.000,E1 280.018} C_DIS
LIN {X 0.016,Y -461.118,Z 301.550,A 0.000,B 0.000,C 90.000,E1 278.973} C_DIS
LIN {X 0.251,Y -469.818,Z 301.541,A 0.000,B 0.000,C 90.000,E1 277.409} C_DIS
LIN {X -0.016,Y -475.220,Z 301.536,A 0.000,B 0.000,C 90.000,E1 276.429} C_DIS
LIN {X -0.086,Y -478.842,Z 301.532,A 0.000,B 0.000,C 90.000,E1 275.682} C_DIS
LIN {X 0.063,Y -480.922,Z 301.529,A 0.000,B 0.000,C 90.000,E1 275.163} C_DIS
LIN {X 0.224,Y -482.706,Z 301.526,A 0.000,B 0.000,C 90.000,E1 274.645} C_DIS
LIN {X -0.129,Y -484.118,Z 301.523,A 0.000,B 0.000,C 90.000,E1 274.188} C_DIS
LIN {X 0.047,Y -485.116,Z 301.520,A 0.000,B 0.000,C 90.000,E1 273.669} C_DIS
LIN {X 0.202,Y -485.740,Z 301.518,A 0.000,B 0.000,C 90.000,E1 273.154} C_DIS
LIN {X -0.096,Y -485.994,Z 301.515,A 0.000,B 0.000,C 90.000,E1 272.694} C_DIS
LIN {X 0.070,Y -485.924,Z 301.512,A 0.000,B 0.000,C 90.000,E1 272.178} C_DIS
LIN {X -0.062,Y -485.133,Z 301.507,A 0.000,B 0.000,C 90.000,E1 271.203} C_DIS
LIN {X 0.106,Y -484.593,Z 301.504,A 0.000,B 0.000,C 90.000,E1 270.688} C_DIS
LIN {X -0.211,Y -483.874,Z 301.501,A 0.000,B 0.000,C 90.000,E1 270.229} C_DIS
LIN {X -0.048,Y -482.797,Z 301.498,A 0.000,B 0.000,C 90.000,E1 269.714} C_DIS
LIN {X 0.110,Y -481.196,Z 301.496,A 0.000,B 0.000,C 90.000,E1 269.198} C_DIS
LIN {X -0.220,Y -479.017,Z 301.493,A 0.000,B 0.000,C 90.000,E1 268.740} C_DIS
LIN {X -0.086,Y -476.064,Z 301.490,A 0.000,B 0.000,C 90.000,E1 268.224} C_DIS
LIN {X 0.227,Y -474.268,Z 301.489,A 0.000,B 0.000,C 90.000,E1 267.936} C_DIS
LIN {X -0.137,Y -469.803,Z 301.486,A 0.000,B 0.000,C 90.000,E1 267.478} C_DIS
LIN {X 0.145,Y -467.144,Z 301.484,A 0.000,B 0.000,C 90.000,E1 267.192} C_DIS
LIN {X 0.057,Y -464.227,Z 301.483,A 0.000,B 0.000,C 90.000,E1 266.963} C_DIS
LIN {X -0.003,Y -460.959,Z 301.482,A 0.000,B 0.000,C 90.000,E1 266.731} C_DIS
LIN {X -0.028,Y -453.983,Z 301.480,A 0.000,B 0.000,C 90.000,E1 266.331} C_DIS
LIN {X 0.143,Y -446.625,Z 301.478,A 0.000,B 0.000,C 90.000,E1 265.988} C_DIS
LIN {X 0.080,Y -442.883,Z 301.477,A 0.000,B 0.000,C 90.000,E1 265.869} C_DIS
LIN {X 0.205,Y -434.289,Z 301.476,A 0.000,B 0.000,C 90.000,E1 265.641} C_DIS
LIN {X 0.078,Y -425.148,Z 301.475,A 0.000,B 0.000,C 90.000,E1 265.527} C_DIS
LIN {X 0.154,Y -417.527,Z 301.475,A 0.000,B 0.000,C 90.000,E1 265.469} C_DIS
LIN {X 0.042,Y -180.907,Z 301.475,A 0.000,B 0.000,C 90.000,E1 265.469} C_DIS
LIN {X 0.094,Y -180.655,Z 301.469,A 0.000,B 0.000,C 90.000,E1 264.432} C_DIS
LIN {X -0.079,Y -179.009,Z 301.445,A 0.000,B 0.000,C 90.000,E1 260.095} C_DIS
LIN {X 0.016,Y -178.623,Z 301.440,A 0.000,B 0.000,C 90.000,E1 259.218} C_DIS
LIN {X -0.085,Y -175.675,Z 301.412,A 0.000,B 0.000,C 90.000,E1 254.157} C_DIS
LIN {X -0.073,Y -172.392,Z 301.388,A 0.000,B 0.000,C 90.000,E1 249.880} C_DIS
LIN {X -0.057,Y -171.196,Z 301.379,A 0.000,B 0.000,C 90.000,E1 248.156} C_DIS
LIN {X -0.006,Y -167.485,Z 301.355,A 0.000,B 0.000,C 90.000,E1 243.819} C_DIS
LIN {X 0.002,Y -166.882,Z 301.350,A 0.000,B 0.000,C 90.000,E1 242.948} C_DIS
LIN {X -0.006,Y -162.187,Z 301.321,A 0.000,B 0.000,C 90.000,E1 237.709} C_DIS
LIN {X -0.039,Y -160.756,Z 301.311,A 0.000,B 0.000,C 90.000,E1 235.960} C_DIS
LIN {X 0.029,Y -157.554,Z 301.291,A 0.000,B 0.000,C 90.000,E1 232.396} C_DIS
LIN {X -0.033,Y -155.582,Z 301.276,A 0.000,B 0.000,C 90.000,E1 229.747} C_DIS
LIN {X 0.019,Y -151.867,Z 301.251,A 0.000,B 0.000,C 90.000,E1 225.243} C_DIS
LIN {X 0.032,Y -150.091,Z 301.236,A 0.000,B 0.000,C 90.000,E1 222.528} C_DIS
LIN {X -0.050,Y -146.892,Z 301.211,A 0.000,B 0.000,C 90.000,E1 218.016} C_DIS
LIN {X 0.055,Y -145.478,Z 301.196,A 0.000,B 0.000,C 90.000,E1 215.231} C_DIS
LIN {X -0.029,Y -142.888,Z 301.170,A 0.000,B 0.000,C 90.000,E1 210.669} C_DIS
LIN {X 0.028,Y -141.508,Z 301.150,A 0.000,B 0.000,C 90.000,E1 206.950} C_DIS
LIN {X -0.054,Y -139.390,Z 301.114,A 0.000,B 0.000,C 90.000,E1 200.482} C_DIS
LIN {X -0.003,Y -139.099,Z 301.103,A 0.000,B 0.000,C 90.000,E1 198.598} C_DIS
LIN {X -0.011,Y -138.353,Z 301.057,A 0.000,B 0.000,C 90.000,E1 190.197} C_DIS
LIN {X -0.018,Y -139.514,Z 301.005,A 0.000,B 0.000,C 90.000,E1 180.859} C_DIS
LIN {X 0.063,Y -141.166,Z 300.974,A 0.000,B 0.000,C 90.000,E1 175.241} C_DIS
LIN {X 0.034,Y -142.546,Z 300.958,A 0.000,B 0.000,C 90.000,E1 172.470} C_DIS
LIN {X -0.040,Y -144.821,Z 300.933,A 0.000,B 0.000,C 90.000,E1 167.881} C_DIS
LIN {X -0.053,Y -147.442,Z 300.912,A 0.000,B 0.000,C 90.000,E1 164.212} C_DIS
LIN {X -0.025,Y -150.023,Z 300.892,A 0.000,B 0.000,C 90.000,E1 160.550} C_DIS
LIN {X -0.018,Y -153.357,Z 300.872,A 0.000,B 0.000,C 90.000,E1 156.922} C_DIS
LIN {X 0.030,Y -155.892,Z 300.857,A 0.000,B 0.000,C 90.000,E1 154.204} C_DIS
LIN {X -0.072,Y -159.750,Z 300.837,A 0.000,B 0.000,C 90.000,E1 150.667} C_DIS
LIN {X -0.006,Y -161.990,Z 300.827,A 0.000,B 0.000,C 90.000,E1 148.869} C_DIS
LIN {X 0.013,Y -166.182,Z 300.807,A 0.000,B 0.000,C 90.000,E1 145.341} C_DIS
LIN {X 0.006,Y -171.196,Z 300.788,A 0.000,B 0.000,C 90.000,E1 141.859} C_DIS
LIN {X 0.036,Y -176.079,Z 300.769,A 0.000,B 0.000,C 90.000,E1 138.405} C_DIS
LIN {X -0.101,Y -180.339,Z 300.755,A 0.000,B 0.000,C 90.000,E1 135.891} C_DIS
LIN {X 0.007,Y -185.749,Z 300.736,A 0.000,B 0.000,C 90.000,E1 132.486} C_DIS
LIN {X -0.080,Y -190.360,Z 300.722,A 0.000,B 0.000,C 90.000,E1 130.011} C_DIS
LIN {X -0.033,Y -197.685,Z 300.699,A 0.000,B 0.000,C 90.000,E1 125.884} C_DIS
LIN {X 0.008,Y -200.936,Z 300.690,A 0.000,B 0.000,C 90.000,E1 124.246} C_DIS
LIN {X 0.046,Y -202.339,Z 300.686,A 0.000,B 0.000,C 90.000,E1 123.420} C_DIS
LIN {X 0.033,Y -304.043,Z 300.686,A 0.000,B 0.000,C 90.000,E1 123.420} C_DIS
LIN {X 0.000,Y -306.642,Z 300.685,A 0.000,B 0.000,C 90.000,E1 123.372} C_DIS
LIN {X 0.120,Y -310.267,Z 300.684,A 0.000,B 0.000,C 90.000,E1 123.166} C_DIS
LIN {X -0.022,Y -312.506,Z 300.683,A 0.000,B 0.000,C 90.000,E1 123.007} C_DIS
LIN {X 0.048,Y -315.624,Z 300.681,A 0.000,B 0.000,C 90.000,E1 122.625} C_DIS
LIN {X -0.129,Y -317.561,Z 300.680,A 0.000,B 0.000,C 90.000,E1 122.339} C_DIS
LIN {X -0.038,Y -319.070,Z 300.678,A 0.000,B 0.000,C 90.000,E1 122.005} C_DIS
LIN {X 0.108,Y -332.644,Z 300.658,A 0.000,B 0.000,C 90.000,E1 118.487} C_DIS
LIN {X -0.061,Y -345.270,Z 300.643,A 0.000,B 0.000,C 90.000,E1 115.720} C_DIS
LIN {X 0.101,Y -357.779,Z 300.629,A 0.000,B 0.000,C 90.000,E1 113.259} C_DIS
LIN {X -0.177,Y -371.597,Z 300.616,A 0.000,B 0.000,C 90.000,E1 110.918} C_DIS
LIN {X 0.115,Y -386.825,Z 300.603,A 0.000,B 0.000,C 90.000,E1 108.544} C_DIS
LIN {X 0.189,Y -403.574,Z 300.590,A 0.000,B 0.000,C 90.000,E1 106.260} C_DIS
LIN {X 0.058,Y -421.970,Z 300.578,A 0.000,B 0.000,C 90.000,E1 104.064} C_DIS
LIN {X -0.008,Y -441.840,Z 300.566,A 0.000,B 0.000,C 90.000,E1 101.951} C_DIS
LIN {X -0.137,Y -462.336,Z 300.556,A 0.000,B 0.000,C 90.000,E1 100.018} C_DIS
LIN {X 0.082,Y -485.982,Z 300.544,A 0.000,B 0.000,C 90.000,E1 97.992} C_DIS
LIN {X -0.080,Y -496.678,Z 300.540,A 0.000,B 0.000,C 90.000,E1 97.182} C_DIS
LIN {X 0.193,Y -499.098,Z 300.539,A 0.000,B 0.000,C 90.000,E1 96.947} C_DIS
LIN {X -0.059,Y -502.542,Z 300.536,A 0.000,B 0.000,C 90.000,E1 96.543} C_DIS
LIN {X -0.197,Y -503.823,Z 300.535,A 0.000,B 0.000,C 90.000,E1 96.315} C_DIS
LIN {X 0.168,Y -504.762,Z 300.534,A 0.000,B 0.000,C 90.000,E1 96.030} C_DIS
LIN {X -0.023,Y -505.775,Z 300.531,A 0.000,B 0.000,C 90.000,E1 95.568} C_DIS
LIN {X -0.212,Y -505.769,Z 300.528,A 0.000,B 0.000,C 90.000,E1 95.106} C_DIS
LIN {X 0.107,Y -504.737,Z 300.526,A 0.000,B 0.000,C 90.000,E1 94.588} C_DIS
LIN {X -0.006,Y -503.787,Z 300.524,A 0.000,B 0.000,C 90.000,E1 94.359} C_DIS
LIN {X -0.117,Y -502.486,Z 300.523,A 0.000,B 0.000,C 90.000,E1 94.131} C_DIS
LIN {X 0.064,Y -497.099,Z 300.519,A 0.000,B 0.000,C 90.000,E1 93.383} C_DIS
LIN {X 0.060,Y -489.095,Z 300.513,A 0.000,B 0.000,C 90.000,E1 92.407} C_DIS
LIN {X -0.057,Y -474.385,Z 300.504,A 0.000,B 0.000,C 90.000,E1 90.688} C_DIS
LIN {X -0.177,Y -454.650,Z 300.490,A 0.000,B 0.000,C 90.000,E1 88.165} C_DIS
LIN {X -0.098,Y -438.629,Z 300.477,A 0.000,B 0.000,C 90.000,E1 85.812} C_DIS
LIN {X 0.180,Y -422.376,Z 300.462,A 0.000,B 0.000,C 90.000,E1 83.109} C_DIS
LIN {X 0.062,Y -403.409,Z 300.442,A 0.000,B 0.000,C 90.000,E1 79.567} C_DIS
LIN {X 0.124,Y -394.773,Z 300.433,A 0.000,B 0.000,C 90.000,E1 77.881} C_DIS
LIN {X -0.144,Y -384.636,Z 300.422,A 0.000,B 0.000,C 90.000,E1 75.936} C_DIS
LIN {X -0.038,Y -373.195,Z 300.409,A 0.000,B 0.000,C 90.000,E1 73.614} C_DIS
LIN {X -0.102,Y -361.654,Z 300.396,A 0.000,B 0.000,C 90.000,E1 71.275} C_DIS
LIN {X 0.115,Y -350.255,Z 300.383,A 0.000,B 0.000,C 90.000,E1 68.847} C_DIS
LIN {X 0.111,Y -337.990,Z 300.367,A 0.000,B 0.000,C 90.000,E1 66.102} C_DIS
LIN {X 0.081,Y -323.502,Z 300.347,A 0.000,B 0.000,C 90.000,E1 62.359} C_DIS
LIN {X 0.078,Y -313.326,Z 300.331,A 0.000,B 0.000,C 90.000,E1 59.488} C_DIS
LIN {X -0.064,Y -305.679,Z 300.318,A 0.000,B 0.000,C 90.000,E1 57.248} C_DIS
LIN {X 0.200,Y -295.393,Z 300.300,A 0.000,B 0.000,C 90.000,E1 53.909} C_DIS
LIN {X -0.013,Y -289.402,Z 300.289,A 0.000,B 0.000,C 90.000,E1 51.949} C_DIS
LIN {X 0.070,Y -283.391,Z 300.277,A 0.000,B 0.000,C 90.000,E1 49.908} C_DIS
LIN {X 0.007,Y -275.369,Z 300.262,A 0.000,B 0.000,C 90.000,E1 47.187} C_DIS
LIN {X 0.044,Y -265.815,Z 300.243,A 0.000,B 0.000,C 90.000,E1 43.704} C_DIS
LIN {X 0.008,Y -260.258,Z 300.231,A 0.000,B 0.000,C 90.000,E1 41.595} C_DIS
LIN {X -0.108,Y -254.607,Z 300.219,A 0.000,B 0.000,C 90.000,E1 39.483} C_DIS
LIN {X 0.061,Y -248.882,Z 300.207,A 0.000,B 0.000,C 90.000,E1 37.282} C_DIS
LIN {X 0.020,Y -243.029,Z 300.195,A 0.000,B 0.000,C 90.000,E1 35.105} C_DIS
LIN {X 0.082,Y -235.063,Z 300.179,A 0.000,B 0.000,C 90.000,E1 32.133} C_DIS
LIN {X -0.025,Y -227.569,Z 300.162,A 0.000,B 0.000,C 90.000,E1 29.155} C_DIS
LIN {X -0.024,Y -220.687,Z 300.145,A 0.000,B 0.000,C 90.000,E1 26.104} C_DIS
LIN {X -0.082,Y -214.601,Z 300.128,A 0.000,B 0.000,C 90.000,E1 23.025} C_DIS
LIN {X -0.056,Y -209.357,Z 300.110,A 0.000,B 0.000,C 90.000,E1 19.885} C_DIS
LIN {X 0.084,Y -204.764,Z 300.093,A 0.000,B 0.000,C 90.000,E1 16.677} C_DIS
LIN {X -0.020,Y -200.024,Z 300.071,A 0.000,B 0.000,C 90.000,E1 12.703} C_DIS
LIN {X 0.097,Y -196.290,Z 300.048,A 0.000,B 0.000,C 90.000,E1 8.624} C_DIS
LIN {X 0.056,Y -192.758,Z 300.016,A 0.000,B 0.000,C 90.000,E1 2.922} C_DIS
LIN {X 0.037,Y -193.431,Z 299.924,A 0.000,B 0.000,C 90.000,E1 346.353} C_DIS
LIN {X -0.002,Y -196.836,Z 299.897,A 0.000,B 0.000,C 90.000,E1 341.456} C_DIS
LIN {X -0.049,Y -200.831,Z 299.874,A 0.000,B 0.000,C 90.000,E1 337.411} C_DIS
LIN {X -0.030,Y -205.870,Z 299.852,A 0.000,B 0.000,C 90.000,E1 333.384} C_DIS
LIN {X -0.037,Y -211.891,Z 299.830,A 0.000,B 0.000,C 90.000,E1 329.410} C_DIS
LIN {X -0.142,Y -217.329,Z 299.813,A 0.000,B 0.000,C 90.000,E1 326.294} C_DIS
LIN {X 0.079,Y -223.523,Z 299.795,A 0.000,B 0.000,C 90.000,E1 323.130} C_DIS
LIN {X 0.060,Y -230.561,Z 299.778,A 0.000,B 0.000,C 90.000,E1 320.070} C_DIS
LIN {X -0.027,Y -239.753,Z 299.759,A 0.000,B 0.000,C 90.000,E1 316.701} C_DIS
LIN {X -0.032,Y -250.189,Z 299.741,A 0.000,B 0.000,C 90.000,E1 313.380} C_DIS
LIN {X 0.133,Y -261.579,Z 299.723,A 0.000,B 0.000,C 90.000,E1 310.092} C_DIS
LIN {X -0.041,Y -274.080,Z 299.705,A 0.000,B 0.000,C 90.000,E1 306.950} C_DIS
LIN {X -0.092,Y -286.288,Z 299.690,A 0.000,B 0.000,C 90.000,E1 304.199} C_DIS
LIN {X 0.092,Y -298.187,Z 299.677,A 0.000,B 0.000,C 90.000,E1 301.799} C_DIS
LIN {X -0.097,Y -315.203,Z 299.660,A 0.000,B 0.000,C 90.000,E1 298.871} C_DIS
LIN {X -0.007,Y -335.936,Z 299.643,A 0.000,B 0.000,C 90.000,E1 295.668} C_DIS
LIN {X -0.063,Y -351.272,Z 299.631,A 0.000,B 0.000,C 90.000,E1 293.515} C_DIS
LIN {X -0.080,Y -366.718,Z 299.619,A 0.000,B 0.000,C 90.000,E1 291.408} C_DIS
LIN {X -0.110,Y -389.292,Z 299.603,A 0.000,B 0.000,C 90.000,E1 288.489} C_DIS
LIN {X -0.239,Y -403.241,Z 299.593,A 0.000,B 0.000,C 90.000,E1 286.804} C_DIS
LIN {X -0.236,Y -417.132,Z 299.584,A 0.000,B 0.000,C 90.000,E1 285.134} C_DIS
LIN {X 0.008,Y -426.288,Z 299.578,A 0.000,B 0.000,C 90.000,E1 284.008} C_DIS
LIN {X 0.192,Y -432.769,Z 299.573,A 0.000,B 0.000,C 90.000,E1 283.175} C_DIS
LIN {X -0.098,Y -438.728,Z 299.569,A 0.000,B 0.000,C 90.000,E1 282.411} C_DIS
LIN {X -0.207,Y -446.170,Z 299.563,A 0.000,B 0.000,C 90.000,E1 281.366} C_DIS
LIN {X -0.139,Y -453.048,Z 299.557,A 0.000,B 0.000,C 90.000,E1 280.310} C_DIS
LIN {X -0.074,Y -459.405,Z 299.551,A 0.000,B 0.000,C 90.000,E1 279.265} C_DIS
LIN {X -0.163,Y -466.779,Z 299.544,A 0.000,B 0.000,C 90.000,E1 277.992} C_DIS
LIN {X -0.150,Y -473.700,Z 299.537,A 0.000,B 0.000,C 90.000,E1 276.720} C_DIS
LIN {X 0.101,Y -478.642,Z 299.532,A 0.000,B 0.000,C 90.000,E1 275.682} C_DIS
LIN {X -0.230,Y -480.782,Z 299.529,A 0.000,B 0.000,C 90.000,E1 275.220} C_DIS
LIN {X -0.071,Y -482.566,Z 299.526,A 0.000,B 0.000,C 90.000,E1 274.702} C_DIS
LIN {X 0.057,Y -483.976,Z 299.523,A 0.000,B 0.000,C 90.000,E1 274.188} C_DIS
LIN {X 0.233,Y -484.971,Z 299.521,A 0.000,B 0.000,C 90.000,E1 273.669} C_DIS
LIN {X -0.099,Y -485.625,Z 299.518,A 0.000,B 0.000,C 90.000,E1 273.212} C_DIS
LIN {X 0.088,Y -485.893,Z 299.515,A 0.000,B 0.000,C 90.000,E1 272.694} C_DIS
LIN {X -0.232,Y -485.828,Z 299.512,A 0.000,B 0.000,C 90.000,E1 272.236} C_DIS
LIN {X 0.121,Y -485.083,Z 299.507,A 0.000,B 0.000,C 90.000,E1 271.203} C_DIS
LIN {X -0.196,Y -484.607,Z 299.504,A 0.000,B 0.000,C 90.000,E1 270.745} C_DIS
LIN {X -0.030,Y -483.865,Z 299.501,A 0.000,B 0.000,C 90.000,E1 270.229} C_DIS
LIN {X 0.132,Y -482.834,Z 299.499,A 0.000,B 0.000,C 90.000,E1 269.714} C_DIS
LIN {X -0.192,Y -481.253,Z 299.496,A 0.000,B 0.000,C 90.000,E1 269.255} C_DIS
LIN {X -0.040,Y -479.098,Z 299.493,A 0.000,B 0.000,C 90.000,E1 268.740} C_DIS
LIN {X 0.098,Y -476.231,Z 299.490,A 0.000,B 0.000,C 90.000,E1 268.224} C_DIS
LIN {X 0.233,Y -472.389,Z 299.487,A 0.000,B 0.000,C 90.000,E1 267.707} C_DIS
LIN {X 0.045,Y -470.085,Z 299.486,A 0.000,B 0.000,C 90.000,E1 267.478} C_DIS
LIN {X -0.229,Y -464.644,Z 299.483,A 0.000,B 0.000,C 90.000,E1 267.020} C_DIS
LIN {X 0.169,Y -461.355,Z 299.482,A 0.000,B 0.000,C 90.000,E1 266.731} C_DIS
LIN {X 0.153,Y -454.646,Z 299.480,A 0.000,B 0.000,C 90.000,E1 266.331} C_DIS
LIN {X -0.189,Y -447.260,Z 299.478,A 0.000,B 0.000,C 90.000,E1 266.045} C_DIS
LIN {X 0.195,Y -443.807,Z 299.477,A 0.000,B 0.000,C 90.000,E1 265.869} C_DIS
LIN {X -0.162,Y -435.608,Z 299.476,A 0.000,B 0.000,C 90.000,E1 265.698} C_DIS
LIN {X 0.015,Y -425.800,Z 299.475,A 0.000,B 0.000,C 90.000,E1 265.527} C_DIS
LIN {X 0.023,Y -417.697,Z 299.475,A 0.000,B 0.000,C 90.000,E1 265.469} C_DIS
LIN {X -0.012,Y -180.906,Z 299.475,A 0.000,B 0.000,C 90.000,E1 265.469} C_DIS
LIN {X 0.066,Y -180.711,Z 299.470,A 0.000,B 0.000,C 90.000,E1 264.552} C_DIS
LIN {X -0.016,Y -178.798,Z 299.442,A 0.000,B 0.000,C 90.000,E1 259.511} C_DIS
LIN {X 0.062,Y -175.844,Z 299.413,A 0.000,B 0.000,C 90.000,E1 254.393} C_DIS
LIN {X 0.061,Y -172.035,Z 299.385,A 0.000,B 0.000,C 90.000,E1 249.263} C_DIS
LIN {X 0.037,Y -171.465,Z 299.380,A 0.000,B 0.000,C 90.000,E1 248.411} C_DIS
LIN {X 0.017,Y -167.696,Z 299.356,A 0.000,B 0.000,C 90.000,E1 244.101} C_DIS
LIN {X 0.031,Y -166.381,Z 299.346,A 0.000,B 0.000,C 90.000,E1 242.359} C_DIS
LIN {X 0.022,Y -163.109,Z 299.327,A 0.000,B 0.000,C 90.000,E1 238.869} C_DIS
LIN {X 0.073,Y -161.057,Z 299.312,A 0.000,B 0.000,C 90.000,E1 236.215} C_DIS
LIN {X -0.040,Y -157.791,Z 299.293,A 0.000,B 0.000,C 90.000,E1 232.718} C_DIS
LIN {X -0.002,Y -155.828,Z 299.278,A 0.000,B 0.000,C 90.000,E1 230.033} C_DIS
LIN {X -0.044,Y -152.078,Z 299.253,A 0.000,B 0.000,C 90.000,E1 225.567} C_DIS
LIN {X -0.025,Y -150.329,Z 299.238,A 0.000,B 0.000,C 90.000,E1 222.852} C_DIS
LIN {X -0.004,Y -147.070,Z 299.213,A 0.000,B 0.000,C 90.000,E1 218.302} C_DIS
LIN {X -0.015,Y -145.644,Z 299.198,A 0.000,B 0.000,C 90.000,E1 215.564} C_DIS
LIN {X -0.095,Y -143.027,Z 299.172,A 0.000,B 0.000,C 90.000,E1 211.003} C_DIS
LIN {X 0.032,Y -141.652,Z 299.151,A 0.000,B 0.000,C 90.000,E1 207.257} C_DIS
LIN {X -0.049,Y -139.444,Z 299.115,A 0.000,B 0.000,C 90.000,E1 200.791} C_DIS
LIN {X 0.003,Y -139.178,Z 299.105,A 0.000,B 0.000,C 90.000,E1 198.906} C_DIS
LIN {X 0.032,Y -138.320,Z 299.053,A 0.000,B 0.000,C 90.000,E1 189.557} C_DIS
LIN {X 0.041,Y -139.468,Z 299.006,A 0.000,B 0.000,C 90.000,E1 181.146} C_DIS
LIN {X -0.018,Y -141.034,Z 298.975,A 0.000,B 0.000,C 90.000,E1 175.584} C_DIS
LIN {X -0.064,Y -142.401,Z 298.960,A 0.000,B 0.000,C 90.000,E1 172.818} C_DIS
LIN {X -0.002,Y -144.634,Z 298.934,A 0.000,B 0.000,C 90.000,E1 168.173} C_DIS
LIN {X 0.059,Y -147.829,Z 298.909,A 0.000,B 0.000,C 90.000,E1 163.559} C_DIS
LIN {X 0.003,Y -150.523,Z 298.889,A 0.000,B 0.000,C 90.000,E1 159.934} C_DIS
LIN {X 0.023,Y -153.986,Z 298.868,A 0.000,B 0.000,C 90.000,E1 156.305} C_DIS
LIN {X -0.057,Y -157.399,Z 298.848,A 0.000,B 0.000,C 90.000,E1 152.743} C_DIS
LIN {X 0.023,Y -161.605,Z 298.829,A 0.000,B 0.000,C 90.000,E1 149.154} C_DIS
LIN {X -0.012,Y -165.802,Z 298.809,A 0.000,B 0.000,C 90.000,E1 145.642} C_DIS
LIN {X 0.015,Y -170.767,Z 298.790,A 0.000,B 0.000,C 90.000,E1 142.145} C_DIS
LIN {X 0.037,Y -175.638,Z 298.771,A 0.000,B 0.000,C 90.000,E1 138.690} C_DIS
LIN {X -0.094,Y -181.253,Z 298.752,A 0.000,B 0.000,C 90.000,E1 135.324} C_DIS
LIN {X 0.036,Y -186.725,Z 298.733,A 0.000,B 0.000,C 90.000,E1 131.919} C_DIS
LIN {X -0.013,Y -191.323,Z 298.719,A 0.000,B 0.000,C 90.000,E1 129.439} C_DIS
LIN {X 0.034,Y -197.156,Z 298.701,A 0.000,B 0.000,C 90.000,E1 126.137} C_DIS
LIN {X -0.047,Y -200.432,Z 298.692,A 0.000,B 0.000,C 90.000,E1 124.532} C_DIS
LIN {X 0.097,Y -202.398,Z 298.686,A 0.000,B 0.000,C 90.000,E1 123.372} C_DIS
LIN {X 0.099,Y -304.242,Z 298.686,A 0.000,B 0.000,C 90.000,E1 123.372} C_DIS
LIN {X -0.127,Y -310.524,Z 298.684,A 0.000,B 0.000,C 90.000,E1 123.166} C_DIS
LIN {X 0.123,Y -313.267,Z 298.683,A 0.000,B 0.000,C 90.000,E1 122.880} C_DIS
LIN {X -0.117,Y -317.016,Z 298.680,A 0.000,B 0.000,C 90.000,E1 122.418} C_DIS
LIN {X -0.057,Y -318.689,Z 298.678,A 0.000,B 0.000,C 90.000,E1 122.084} C_DIS
LIN {X -0.026,Y -323.520,Z 298.671,A 0.000,B 0.000,C 90.000,E1 120.797} C_DIS
LIN {X -0.141,Y -334.991,Z 298.655,A 0.000,B 0.000,C 90.000,E1 117.975} C_DIS
LIN {X 0.067,Y -347.907,Z 298.640,A 0.000,B 0.000,C 90.000,E1 115.155} C_DIS
LIN {X -0.169,Y -360.697,Z 298.626,A 0.000,B 0.000,C 90.000,E1 112.770} C_DIS
LIN {X -0.029,Y -374.818,Z 298.613,A 0.000,B 0.000,C 90.000,E1 110.375} C_DIS
LIN {X -0.013,Y -390.371,Z 298.600,A 0.000,B 0.000,C 90.000,E1 108.055} C_DIS
LIN {X 0.026,Y -407.473,Z 298.588,A 0.000,B 0.000,C 90.000,E1 105.788} C_DIS
LIN {X -0.013,Y -426.251,Z 298.576,A 0.000,B 0.000,C 90.000,E1 103.592} C_DIS
LIN {X 0.200,Y -446.294,Z 298.564,A 0.000,B 0.000,C 90.000,E1 101.478} C_DIS
LIN {X -0.168,Y -466.908,Z 298.553,A 0.000,B 0.000,C 90.000,E1 99.613} C_DIS
LIN {X -0.131,Y -490.697,Z 298.542,A 0.000,B 0.000,C 90.000,E1 97.644} C_DIS
LIN {X 0.101,Y -498.621,Z 298.539,A 0.000,B 0.000,C 90.000,E1 97.004} C_DIS
LIN {X -0.168,Y -500.613,Z 298.538,A 0.000,B 0.000,C 90.000,E1 96.834} C_DIS
LIN {X 0.200,Y -502.433,Z 298.536,A 0.000,B 0.000,C 90.000,E1 96.549} C_DIS
LIN {X 0.126,Y -503.802,Z 298.535,A 0.000,B 0.000,C 90.000,E1 96.315} C_DIS
LIN {X -0.075,Y -505.520,Z 298.532,A 0.000,B 0.000,C 90.000,E1 95.853} C_DIS
LIN {X 0.233,Y -506.137,Z 298.530,A 0.000,B 0.000,C 90.000,E1 95.334} C_DIS
LIN {X 0.002,Y -505.751,Z 298.527,A 0.000,B 0.000,C 90.000,E1 94.878} C_DIS
LIN {X -0.180,Y -504.292,Z 298.524,A 0.000,B 0.000,C 90.000,E1 94.416} C_DIS
LIN {X 0.211,Y -503.080,Z 298.523,A 0.000,B 0.000,C 90.000,E1 94.131} C_DIS
LIN {X 0.017,Y -499.660,Z 298.520,A 0.000,B 0.000,C 90.000,E1 93.669} C_DIS
LIN {X 0.040,Y -491.870,Z 298.515,A 0.000,B 0.000,C 90.000,E1 92.694} C_DIS
LIN {X -0.179,Y -481.431,Z 298.508,A 0.000,B 0.000,C 90.000,E1 91.489} C_DIS
LIN {X 0.085,Y -462.968,Z 298.496,A 0.000,B 0.000,C 90.000,E1 89.198} C_DIS
LIN {X 0.135,Y -447.935,Z 298.484,A 0.000,B 0.000,C 90.000,E1 87.135} C_DIS
LIN {X -0.046,Y -429.236,Z 298.468,A 0.000,B 0.000,C 90.000,E1 84.261} C_DIS
LIN {X 0.055,Y -413.877,Z 298.453,A 0.000,B 0.000,C 90.000,E1 81.546} C_DIS
LIN {X 0.046,Y -402.479,Z 298.441,A 0.000,B 0.000,C 90.000,E1 79.342} C_DIS
LIN {X 0.166,Y -393.821,Z 298.431,A 0.000,B 0.000,C 90.000,E1 77.645} C_DIS
LIN {X -0.160,Y -385.135,Z 298.422,A 0.000,B 0.000,C 90.000,E1 75.992} C_DIS
LIN {X -0.141,Y -373.690,Z 298.409,A 0.000,B 0.000,C 90.000,E1 73.685} C_DIS
LIN {X -0.165,Y -363.609,Z 298.398,A 0.000,B 0.000,C 90.000,E1 71.638} C_DIS
LIN {X 0.104,Y -352.196,Z 298.385,A 0.000,B 0.000,C 90.000,E1 69.209} C_DIS
LIN {X 0.027,Y -337.264,Z 298.366,A 0.000,B 0.000,C 90.000,E1 65.869} C_DIS
LIN {X 0.010,Y -324.026,Z 298.347,A 0.000,B 0.000,C 90.000,E1 62.436} C_DIS
LIN {X 0.107,Y -314.944,Z 298.333,A 0.000,B 0.000,C 90.000,E1 59.871} C_DIS
LIN {X -0.154,Y -307.289,Z 298.320,A 0.000,B 0.000,C 90.000,E1 57.661} C_DIS
LIN {X -0.010,Y -296.909,Z 298.302,A 0.000,B 0.000,C 90.000,E1 54.356} C_DIS
LIN {X -0.055,Y -288.898,Z 298.287,A 0.000,B 0.000,C 90.000,E1 51.698} C_DIS
LIN {X 0.025,Y -280.823,Z 298.272,A 0.000,B 0.000,C 90.000,E1 48.976} C_DIS
LIN {X -0.125,Y -270.933,Z 298.253,A 0.000,B 0.000,C 90.000,E1 45.567} C_DIS
LIN {X -0.132,Y -263.459,Z 298.237,A 0.000,B 0.000,C 90.000,E1 42.771} C_DIS
LIN {X -0.015,Y -257.856,Z 298.226,A 0.000,B 0.000,C 90.000,E1 40.620} C_DIS
LIN {X 0.022,Y -252.203,Z 298.214,A 0.000,B 0.000,C 90.000,E1 38.463} C_DIS
LIN {X -0.007,Y -246.410,Z 298.202,A 0.000,B 0.000,C 90.000,E1 36.297} C_DIS
LIN {X -0.090,Y -240.462,Z 298.189,A 0.000,B 0.000,C 90.000,E1 34.119} C_DIS
LIN {X -0.036,Y -230.710,Z 298.169,A 0.000,B 0.000,C 90.000,E1 30.384} C_DIS
LIN {X 0.040,Y -223.596,Z 298.152,A 0.000,B 0.000,C 90.000,E1 27.334} C_DIS
LIN {X 0.036,Y -217.230,Z 298.135,A 0.000,B 0.000,C 90.000,E1 24.259} C_DIS
LIN {X -0.002,Y -211.615,Z 298.118,A 0.000,B 0.000,C 90.000,E1 21.153} C_DIS
LIN {X -0.057,Y -205.674,Z 298.096,A 0.000,B 0.000,C 90.000,E1 17.221} C_DIS
LIN {X 0.117,Y -200.792,Z 298.073,A 0.000,B 0.000,C 90.000,E1 13.175} C_DIS
LIN {X 0.065,Y -196.931,Z 298.051,A 0.000,B 0.000,C 90.000,E1 9.151} C_DIS
LIN {X -0.065,Y -193.643,Z 298.024,A 0.000,B 0.000,C 90.000,E1 4.302} C_DIS
LIN {X -0.046,Y -191.280,Z 297.984,A 0.000,B 0.000,C 90.000,E1 357.078} C_DIS
LIN {X 0.060,Y -192.776,Z 297.933,A 0.000,B 0.000,C 90.000,E1 347.993} C_DIS
LIN {X -0.099,Y -196.296,Z 297.902,A 0.000,B 0.000,C 90.000,E1 342.308} C_DIS
LIN {X -0.056,Y -200.085,Z 297.879,A 0.000,B 0.000,C 90.000,E1 338.230} C_DIS
LIN {X -0.065,Y -204.904,Z 297.857,A 0.000,B 0.000,C 90.000,E1 334.204} C_DIS
LIN {X -0.015,Y -210.733,Z 297.834,A 0.000,B 0.000,C 90.000,E1 330.205} C_DIS
LIN {X -0.100,Y -217.433,Z 297.813,A 0.000,B 0.000,C 90.000,E1 326.294} C_DIS
LIN {X 0.126,Y -223.661,Z 297.795,A 0.000,B 0.000,C 90.000,E1 323.130} C_DIS
LIN {X -0.065,Y -230.731,Z 297.778,A 0.000,B 0.000,C 90.000,E1 320.114} C_DIS
LIN {X 0.033,Y -239.947,Z 297.759,A 0.000,B 0.000,C 90.000,E1 316.701} C_DIS
LIN {X 0.037,Y -250.377,Z 297.741,A 0.000,B 0.000,C 90.000,E1 313.380} C_DIS
LIN {X -0.159,Y -261.766,Z 297.723,A 0.000,B 0.000,C 90.000,E1 310.172} C_DIS
LIN {X 0.044,Y -274.259,Z 297.705,A 0.000,B 0.000,C 90.000,E1 306.950} C_DIS
LIN {X 0.002,Y -286.485,Z 297.690,A 0.000,B 0.000,C 90.000,E1 304.199} C_DIS
LIN {X -0.058,Y -300.180,Z 297.675,A 0.000,B 0.000,C 90.000,E1 301.514} C_DIS
LIN {X -0.075,Y -317.423,Z 297.659,A 0.000,B 0.000,C 90.000,E1 298.565} C_DIS
LIN {X -0.057,Y -338.317,Z 297.641,A 0.000,B 0.000,C 90.000,E1 295.387} C_DIS
LIN {X 0.078,Y -351.484,Z 297.631,A 0.000,B 0.000,C 90.000,E1 293.515} C_DIS
LIN {X 0.072,Y -366.877,Z 297.619,A 0.000,B 0.000,C 90.000,E1 291.408} C_DIS
LIN {X 0.056,Y -389.378,Z 297.603,A 0.000,B 0.000,C 90.000,E1 288.489} C_DIS
LIN {X -0.065,Y -403.263,Z 297.593,A 0.000,B 0.000,C 90.000,E1 286.804} C_DIS
LIN {X 0.180,Y -419.416,Z 297.583,A 0.000,B 0.000,C 90.000,E1 284.828} C_DIS
LIN {X -0.062,Y -428.396,Z 297.576,A 0.000,B 0.000,C 90.000,E1 283.772} C_DIS
LIN {X 0.132,Y -434.684,Z 297.572,A 0.000,B 0.000,C 90.000,E1 282.939} C_DIS
LIN {X 0.068,Y -442.399,Z 297.566,A 0.000,B 0.000,C 90.000,E1 281.883} C_DIS
LIN {X 0.006,Y -449.531,Z 297.560,A 0.000,B 0.000,C 90.000,E1 280.838} C_DIS
LIN {X -0.150,Y -457.688,Z 297.553,A 0.000,B 0.000,C 90.000,E1 279.557} C_DIS
LIN {X -0.201,Y -465.120,Z 297.546,A 0.000,B 0.000,C 90.000,E1 278.276} C_DIS
LIN {X 0.254,Y -472.139,Z 297.539,A 0.000,B 0.000,C 90.000,E1 276.947} C_DIS
LIN {X 0.012,Y -477.271,Z 297.533,A 0.000,B 0.000,C 90.000,E1 275.967} C_DIS
LIN {X -0.041,Y -480.593,Z 297.529,A 0.000,B 0.000,C 90.000,E1 275.220} C_DIS
LIN {X 0.117,Y -482.396,Z 297.526,A 0.000,B 0.000,C 90.000,E1 274.702} C_DIS
LIN {X -0.238,Y -483.834,Z 297.523,A 0.000,B 0.000,C 90.000,E1 274.245} C_DIS
LIN {X -0.063,Y -484.875,Z 297.521,A 0.000,B 0.000,C 90.000,E1 273.726} C_DIS
LIN {X 0.089,Y -485.534,Z 297.518,A 0.000,B 0.000,C 90.000,E1 273.212} C_DIS
LIN {X -0.211,Y -485.802,Z 297.515,A 0.000,B 0.000,C 90.000,E1 272.751} C_DIS
LIN {X -0.046,Y -485.749,Z 297.512,A 0.000,B 0.000,C 90.000,E1 272.236} C_DIS
LIN {X -0.180,Y -485.020,Z 297.507,A 0.000,B 0.000,C 90.000,E1 271.260} C_DIS
LIN {X -0.013,Y -484.549,Z 297.504,A 0.000,B 0.000,C 90.000,E1 270.745} C_DIS
LIN {X 0.153,Y -483.863,Z 297.501,A 0.000,B 0.000,C 90.000,E1 270.229} C_DIS
LIN {X -0.168,Y -482.841,Z 297.499,A 0.000,B 0.000,C 90.000,E1 269.771} C_DIS
LIN {X -0.010,Y -481.290,Z 297.496,A 0.000,B 0.000,C 90.000,E1 269.255} C_DIS
LIN {X 0.141,Y -479.186,Z 297.493,A 0.000,B 0.000,C 90.000,E1 268.740} C_DIS
LIN {X -0.196,Y -476.339,Z 297.490,A 0.000,B 0.000,C 90.000,E1 268.282} C_DIS
LIN {X 0.116,Y -474.596,Z 297.489,A 0.000,B 0.000,C 90.000,E1 267.993} C_DIS
LIN {X 0.224,Y -470.286,Z 297.486,A 0.000,B 0.000,C 90.000,E1 267.478} C_DIS
LIN {X -0.076,Y -464.920,Z 297.483,A 0.000,B 0.000,C 90.000,E1 267.020} C_DIS
LIN {X 0.036,Y -458.620,Z 297.481,A 0.000,B 0.000,C 90.000,E1 266.560} C_DIS
LIN {X -0.223,Y -455.030,Z 297.480,A 0.000,B 0.000,C 90.000,E1 266.388} C_DIS
LIN {X -0.128,Y -447.889,Z 297.478,A 0.000,B 0.000,C 90.000,E1 266.045} C_DIS
LIN {X 0.207,Y -444.318,Z 297.477,A 0.000,B 0.000,C 90.000,E1 265.869} C_DIS
LIN {X 0.066,Y -439.955,Z 297.476,A 0.000,B 0.000,C 90.000,E1 265.755} C_DIS
LIN {X 0.216,Y -435.997,Z 297.476,A 0.000,B 0.000,C 90.000,E1 265.641} C_DIS
LIN {X -0.068,Y -426.794,Z 297.475,A 0.000,B 0.000,C 90.000,E1 265.527} C_DIS
LIN {X -0.067,Y -419.132,Z 297.475,A 0.000,B 0.000,C 90.000,E1 265.469} C_DIS
LIN {X -0.053,Y -180.906,Z 297.475,A 0.000,B 0.000,C 90.000,E1 265.469} C_DIS
LIN {X 0.031,Y -180.703,Z 297.470,A 0.000,B 0.000,C 90.000,E1 264.546} C_DIS
LIN {X -0.068,Y -178.789,Z 297.442,A 0.000,B 0.000,C 90.000,E1 259.511} C_DIS
LIN {X 0.009,Y -175.835,Z 297.413,A 0.000,B 0.000,C 90.000,E1 254.393} C_DIS
LIN {X 0.010,Y -172.024,Z 297.385,A 0.000,B 0.000,C 90.000,E1 249.263} C_DIS
LIN {X -0.013,Y -171.450,Z 297.380,A 0.000,B 0.000,C 90.000,E1 248.411} C_DIS
LIN {X 0.040,Y -167.684,Z 297.356,A 0.000,B 0.000,C 90.000,E1 244.076} C_DIS
LIN {X -0.019,Y -166.363,Z 297.346,A 0.000,B 0.000,C 90.000,E1 242.359} C_DIS
LIN {X -0.027,Y -163.094,Z 297.327,A 0.000,B 0.000,C 90.000,E1 238.869} C_DIS
LIN {X 0.023,Y -161.039,Z 297.312,A 0.000,B 0.000,C 90.000,E1 236.215} C_DIS
LIN {X 0.007,Y -157.778,Z 297.293,A 0.000,B 0.000,C 90.000,E1 232.683} C_DIS
LIN {X 0.070,Y -155.815,Z 297.278,A 0.000,B 0.000,C 90.000,E1 229.989} C_DIS
LIN {X 0.017,Y -152.066,Z 297.253,A 0.000,B 0.000,C 90.000,E1 225.526} C_DIS
LIN {X -0.072,Y -150.316,Z 297.238,A 0.000,B 0.000,C 90.000,E1 222.852} C_DIS
LIN {X -0.050,Y -147.059,Z 297.213,A 0.000,B 0.000,C 90.000,E1 218.302} C_DIS
LIN {X 0.057,Y -145.636,Z 297.197,A 0.000,B 0.000,C 90.000,E1 215.518} C_DIS
LIN {X 0.055,Y -143.019,Z 297.172,A 0.000,B 0.000,C 90.000,E1 210.924} C_DIS
LIN {X -0.013,Y -141.645,Z 297.151,A 0.000,B 0.000,C 90.000,E1 207.257} C_DIS
LIN {X 0.037,Y -139.441,Z 297.115,A 0.000,B 0.000,C 90.000,E1 200.737} C_DIS
LIN {X -0.041,Y -139.174,Z 297.105,A 0.000,B 0.000,C 90.000,E1 198.906} C_DIS
LIN {X -0.013,Y -138.318,Z 297.053,A 0.000,B 0.000,C 90.000,E1 189.557} C_DIS
LIN {X -0.004,Y -139.471,Z 297.006,A 0.000,B 0.000,C 90.000,E1 181.146} C_DIS
LIN {X -0.064,Y -141.042,Z 296.975,A 0.000,B 0.000,C 90.000,E1 175.584} C_DIS
LIN {X 0.032,Y -142.411,Z 296.960,A 0.000,B 0.000,C 90.000,E1 172.761} C_DIS
LIN {X -0.048,Y -144.645,Z 296.934,A 0.000,B 0.000,C 90.000,E1 168.173} C_DIS
LIN {X 0.011,Y -147.841,Z 296.909,A 0.000,B 0.000,C 90.000,E1 163.559} C_DIS
LIN {X -0.045,Y -150.539,Z 296.888,A 0.000,B 0.000,C 90.000,E1 159.934} C_DIS
LIN {X -0.025,Y -154.004,Z 296.868,A 0.000,B 0.000,C 90.000,E1 156.305} C_DIS
LIN {X 0.034,Y -157.418,Z 296.848,A 0.000,B 0.000,C 90.000,E1 152.692} C_DIS
LIN {X 0.057,Y -161.628,Z 296.829,A 0.000,B 0.000,C 90.000,E1 149.125} C_DIS
LIN {X 0.075,Y -165.825,Z 296.809,A 0.000,B 0.000,C 90.000,E1 145.595} C_DIS
LIN {X 0.068,Y -170.793,Z 296.790,A 0.000,B 0.000,C 90.000,E1 142.110} C_DIS
LIN {X -0.015,Y -175.664,Z 296.770,A 0.000,B 0.000,C 90.000,E1 138.690} C_DIS
LIN {X -0.018,Y -181.278,Z 296.752,A 0.000,B 0.000,C 90.000,E1 135.283} C_DIS
LIN {X -0.018,Y -186.755,Z 296.733,A 0.000,B 0.000,C 90.000,E1 131.919} C_DIS
LIN {X 0.054,Y -191.350,Z 296.719,A 0.000,B 0.000,C 90.000,E1 129.402} C_DIS
LIN {X -0.021,Y -197.187,Z 296.701,A 0.000,B 0.000,C 90.000,E1 126.137} C_DIS
LIN {X 0.062,Y -200.465,Z 296.692,A 0.000,B 0.000,C 90.000,E1 124.485} C_DIS
LIN {X -0.023,Y -202.459,Z 296.685,A 0.000,B 0.000,C 90.000,E1 123.372} C_DIS
LIN {X -0.070,Y -303.726,Z 296.685,A 0.000,B 0.000,C 90.000,E1 123.372} C_DIS
LIN {X 0.068,Y -306.713,Z 296.685,A 0.000,B 0.000,C 90.000,E1 123.293} C_DIS
LIN {X 0.051,Y -310.755,Z 296.684,A 0.000,B 0.000,C 90.000,E1 123.086} C_DIS
LIN {X 0.036,Y -313.166,Z 296.683,A 0.000,B 0.000,C 90.000,E1 122.880} C_DIS
LIN {X -0.194,Y -316.983,Z 296.680,A 0.000,B 0.000,C 90.000,E1 122.418} C_DIS
LIN {X -0.134,Y -318.690,Z 296.678,A 0.000,B 0.000,C 90.000,E1 122.084} C_DIS
LIN {X 0.086,Y -322.361,Z 296.673,A 0.000,B 0.000,C 90.000,E1 121.082} C_DIS
LIN {X 0.112,Y -333.682,Z 296.657,A 0.000,B 0.000,C 90.000,E1 118.231} C_DIS
LIN {X -0.027,Y -346.442,Z 296.641,A 0.000,B 0.000,C 90.000,E1 115.463} C_DIS
LIN {X 0.024,Y -359.080,Z 296.628,A 0.000,B 0.000,C 90.000,E1 113.025} C_DIS
LIN {X -0.083,Y -373.036,Z 296.615,A 0.000,B 0.000,C 90.000,E1 110.663} C_DIS
LIN {X 0.120,Y -388.413,Z 296.602,A 0.000,B 0.000,C 90.000,E1 108.308} C_DIS
LIN {X -0.151,Y -405.323,Z 296.589,A 0.000,B 0.000,C 90.000,E1 106.079} C_DIS
LIN {X 0.156,Y -423.895,Z 296.577,A 0.000,B 0.000,C 90.000,E1 103.828} C_DIS
LIN {X -0.222,Y -443.858,Z 296.565,A 0.000,B 0.000,C 90.000,E1 101.771} C_DIS
LIN {X 0.147,Y -464.409,Z 296.555,A 0.000,B 0.000,C 90.000,E1 99.792} C_DIS
LIN {X 0.124,Y -488.108,Z 296.543,A 0.000,B 0.000,C 90.000,E1 97.814} C_DIS
LIN {X 0.017,Y -498.738,Z 296.539,A 0.000,B 0.000,C 90.000,E1 97.004} C_DIS
LIN {X 0.246,Y -500.761,Z 296.538,A 0.000,B 0.000,C 90.000,E1 96.777} C_DIS
LIN {X 0.136,Y -502.594,Z 296.536,A 0.000,B 0.000,C 90.000,E1 96.549} C_DIS
LIN {X 0.081,Y -503.976,Z 296.535,A 0.000,B 0.000,C 90.000,E1 96.315} C_DIS
LIN {X -0.120,Y -505.738,Z 296.532,A 0.000,B 0.000,C 90.000,E1 95.853} C_DIS
LIN {X 0.190,Y -506.391,Z 296.530,A 0.000,B 0.000,C 90.000,E1 95.334} C_DIS
LIN {X -0.040,Y -506.037,Z 296.527,A 0.000,B 0.000,C 90.000,E1 94.878} C_DIS
LIN {X -0.220,Y -504.617,Z 296.524,A 0.000,B 0.000,C 90.000,E1 94.416} C_DIS
LIN {X 0.172,Y -503.428,Z 296.523,A 0.000,B 0.000,C 90.000,E1 94.131} C_DIS
LIN {X -0.020,Y -499.984,Z 296.520,A 0.000,B 0.000,C 90.000,E1 93.669} C_DIS
